C01827=1158.573,334.839,-76.760,-176.548,8.692,148.725
C01828=1158.569,335.087,-76.793,-176.546,8.695,148.726
C01829=1158.565,335.335,-76.827,-176.543,8.698,148.726
C01830=1158.562,335.582,-76.859,-176.540,8.702,148.726
C01831=1158.557,335.831,-76.892,-176.538,8.706,148.726
C01832=1158.553,336.078,-76.925,-176.536,8.709,148.726
C01833=1158.549,336.326,-76.958,-176.532,8.713,148.727
C01834=1158.545,336.574,-76.991,-176.530,8.716,148.727
C01835=1158.541,336.822,-77.024,-176.528,8.719,148.727
C01836=1158.537,337.069,-77.057,-176.525,8.723,148.727
C01837=1158.532,337.317,-77.091,-176.523,8.727,148.727
C01838=1158.529,337.565,-77.124,-176.520,8.730,148.728
C01839=1158.525,337.813,-77.157,-176.517,8.734,148.728
C01840=1158.521,338.061,-77.190,-176.515,8.737,148.728
C01841=1158.516,338.309,-77.224,-176.513,8.741,148.728
C01842=1158.512,338.556,-77.257,-176.510,8.745,148.728
C01843=1158.509,338.804,-77.291,-176.508,8.748,148.729
C01844=1158.504,339.051,-77.324,-176.505,8.751,148.729
C01845=1158.500,339.331,-77.361,-176.502,8.755,148.729
C01846=1158.495,339.612,-77.398,-176.500,8.759,148.729
C01847=1158.491,339.891,-77.436,-176.497,8.764,148.730
C01848=1158.486,340.171,-77.473,-176.494,8.768,148.730
C01849=1158.482,340.418,-77.508,-176.491,8.771,148.730
C01850=1158.478,340.666,-77.541,-176.489,8.775,148.730
C01851=1158.473,340.914,-77.574,-176.486,8.778,148.731
C01852=1158.469,341.162,-77.607,-176.484,8.782,148.731
C01853=1158.466,341.410,-77.641,-176.482,8.786,148.731
C01854=1158.462,341.657,-77.675,-176.479,8.789,148.731
C01855=1158.458,341.905,-77.708,-176.476,8.793,148.732
C01856=1158.454,342.153,-77.741,-176.474,8.797,148.732
C01857=1158.449,342.401,-77.775,-176.472,8.800,148.732
C01858=1158.445,342.648,-77.809,-176.469,8.804,148.732
C01859=1158.441,342.896,-77.842,-176.467,8.807,148.733
C01860=1158.437,343.144,-77.875,-176.464,8.811,148.733
C01861=1158.433,343.391,-77.909,-176.461,8.815,148.733
C01862=1158.429,343.639,-77.942,-176.459,8.818,148.733
C01863=1158.424,343.887,-77.976,-176.456,8.822,148.733
C01864=1158.421,344.135,-78.010,-176.454,8.825,148.734
C01865=1158.417,344.382,-78.044,-176.452,8.829,148.734
C01866=1158.413,344.629,-78.077,-176.449,8.833,148.734
C01867=1158.408,344.877,-78.111,-176.446,8.836,148.734
C01868=1158.405,345.124,-78.145,-176.444,8.841,148.735
C01869=1158.401,345.373,-78.179,-176.442,8.844,148.735
C01870=1158.397,345.621,-78.212,-176.439,8.847,148.735
C01871=1158.392,345.868,-78.246,-176.436,8.851,148.736
C01872=1158.388,346.116,-78.279,-176.434,8.854,148.736
C01873=1158.385,346.364,-78.314,-176.431,8.859,148.736
C01874=1158.381,346.611,-78.348,-176.429,8.862,148.736
C01875=1158.376,346.859,-78.381,-176.427,8.865,148.736
C01876=1158.372,347.106,-78.415,-176.424,8.869,148.737
C01877=1158.369,347.354,-78.449,-176.422,8.873,148.737
C01878=1158.364,347.602,-78.483,-176.419,8.877,148.737
C01879=1158.360,347.849,-78.516,-176.417,8.880,148.738
C01880=1158.357,348.097,-78.551,-176.414,8.884,148.738
C01881=1158.352,348.345,-78.585,-176.411,8.888,148.738
C01882=1158.348,348.592,-78.618,-176.409,8.891,148.738
C01883=1158.344,348.840,-78.652,-176.407,8.895,148.739
C01884=1158.340,349.088,-78.687,-176.404,8.899,148.739
C01885=1158.336,349.335,-78.720,-176.402,8.902,148.739
C01886=1158.332,349.583,-78.754,-176.399,8.906,148.739
C01887=1158.328,349.831,-78.789,-176.397,8.909,148.740
C01888=1158.324,350.078,-78.822,-176.394,8.913,148.740
C01889=1158.320,350.326,-78.856,-176.392,8.917,148.740
C01890=1158.316,350.574,-78.891,-176.389,8.921,148.740
C01891=1158.312,350.821,-78.925,-176.387,8.924,148.741
C01892=1158.308,351.068,-78.959,-176.385,8.928,148.741
C01893=1158.304,351.317,-78.993,-176.382,8.932,148.741
C01894=1158.300,351.564,-79.027,-176.380,8.935,148.742
C01895=1158.296,351.812,-79.062,-176.377,8.939,148.742
C01896=1158.292,352.059,-79.096,-176.375,8.943,148.742
C01897=1158.288,352.307,-79.130,-176.372,8.947,148.742
C01898=1158.284,352.554,-79.164,-176.369,8.950,148.743
C01899=1158.280,352.802,-79.199,-176.367,8.955,148.743
C01900=1158.276,353.050,-79.232,-176.365,8.958,148.743
C01901=1158.272,353.298,-79.267,-176.362,8.962,148.743
C01902=1158.268,353.545,-79.301,-176.359,8.965,148.744
C01903=1158.264,353.793,-79.335,-176.358,8.969,148.744
C01904=1158.260,354.040,-79.369,-176.355,8.973,148.744
C01905=1158.256,354.288,-79.404,-176.352,8.976,148.745
C01906=1158.252,354.535,-79.438,-176.350,8.980,148.745
C01907=1158.248,354.783,-79.473,-176.348,8.984,148.745
C01908=1158.244,355.031,-79.507,-176.345,8.988,148.746
C01909=1158.240,355.278,-79.541,-176.342,8.991,148.746
C01910=1158.236,355.526,-79.576,-176.340,8.995,148.746
C01911=1158.232,355.773,-79.610,-176.338,8.999,148.746
C01912=1158.228,356.021,-79.645,-176.335,9.003,148.747
C01913=1158.224,356.268,-79.680,-176.333,9.006,148.747
C01914=1158.221,356.516,-79.714,-176.330,9.011,148.747
C01915=1158.216,356.763,-79.749,-176.328,9.014,148.748
C01916=1158.212,357.011,-79.783,-176.325,9.018,148.748
C01917=1158.208,357.258,-79.817,-176.323,9.021,148.748
C01918=1158.204,357.507,-79.852,-176.320,9.026,148.749
C01919=1158.200,357.754,-79.887,-176.318,9.029,148.749
C01920=1158.197,358.001,-79.922,-176.315,9.033,148.749
C01921=1158.192,358.249,-79.956,-176.313,9.037,148.749
C01922=1158.188,358.497,-79.991,-176.310,9.041,148.750
C01923=1158.184,358.744,-80.025,-176.308,9.044,148.750
C01924=1158.181,358.991,-80.060,-176.305,9.049,148.750
C01925=1158.177,359.239,-80.095,-176.303,9.052,148.751
C01926=1158.172,359.487,-80.130,-176.300,9.056,148.751
C01927=1158.169,359.735,-80.164,-176.298,9.060,148.751
C01928=1158.165,359.982,-80.199,-176.295,9.064,148.752
C01929=1158.161,360.230,-80.234,-176.293,9.067,148.752
C01930=1158.156,360.477,-80.268,-176.291,9.071,148.752
C01931=1158.153,360.724,-80.303,-176.288,9.075,148.752
C01932=1158.149,360.972,-80.338,-176.285,9.079,148.753
C01933=1158.145,361.219,-80.373,-176.283,9.083,148.753
C01934=1158.141,361.467,-80.408,-176.281,9.086,148.753
C01935=1158.137,361.715,-80.443,-176.278,9.091,148.754
C01936=1158.133,361.962,-80.478,-176.276,9.094,148.754
C01937=1158.130,362.210,-80.512,-176.273,9.098,148.754
C01938=1158.125,362.457,-80.548,-176.271,9.103,148.755
C01939=1158.121,362.705,-80.582,-176.268,9.106,148.755
C01940=1158.117,362.952,-80.618,-176.266,9.110,148.756
C01941=1158.113,363.200,-80.652,-176.263,9.114,148.756
C01942=1158.109,363.447,-80.688,-176.261,9.118,148.756
C01943=1158.105,363.695,-80.722,-176.259,9.121,148.756
C01944=1158.102,363.942,-80.757,-176.256,9.125,148.757
C01945=1158.098,364.190,-80.792,-176.253,9.130,148.757
C01946=1158.094,364.437,-80.827,-176.251,9.133,148.757
C01947=1158.090,364.684,-80.863,-176.249,9.138,148.758
C01948=1158.086,364.933,-80.898,-176.246,9.141,148.758
C01949=1158.081,365.215,-80.938,-176.243,9.146,148.759
C01950=1158.077,365.498,-80.978,-176.241,9.150,148.759
C01951=1158.072,365.781,-81.019,-176.238,9.155,148.759
C01952=1158.068,366.063,-81.059,-176.235,9.159,148.760
C01953=1158.064,366.311,-81.094,-176.233,9.163,148.760
C01954=1158.060,366.558,-81.129,-176.231,9.167,148.761
C01955=1158.056,366.806,-81.164,-176.228,9.171,148.761
C01956=1158.053,367.053,-81.200,-176.226,9.175,148.761
C01957=1158.048,367.300,-81.235,-176.223,9.179,148.762
C01958=1158.044,367.548,-81.270,-176.221,9.183,148.762
C01959=1158.041,367.796,-81.305,-176.219,9.187,148.763
C01960=1158.037,368.043,-81.341,-176.216,9.191,148.763
C01961=1158.033,368.290,-81.376,-176.214,9.194,148.763
C01962=1158.029,368.537,-81.412,-176.212,9.199,148.764
C01963=1158.024,368.786,-81.447,-176.210,9.202,148.764
C01964=1158.021,369.033,-81.482,-176.208,9.207,148.765
C01965=1158.016,369.280,-81.518,-176.206,9.210,148.765
C01966=1158.013,369.528,-81.553,-176.203,9.215,148.765
C01967=1158.009,369.775,-81.589,-176.201,9.218,148.766
C01968=1158.005,370.023,-81.624,-176.198,9.223,148.766
C01969=1158.001,370.269,-81.660,-176.197,9.226,148.767
C01970=1157.998,370.517,-81.695,-176.194,9.231,148.767
C01971=1157.993,370.765,-81.731,-176.192,9.234,148.768
C01972=1157.989,371.013,-81.766,-176.190,9.238,148.768
C01973=1157.986,371.260,-81.802,-176.188,9.242,148.768
C01974=1157.981,371.507,-81.837,-176.186,9.246,148.769
C01975=1157.978,371.755,-81.872,-176.184,9.250,148.770
C01976=1157.974,372.002,-81.908,-176.182,9.254,148.770
C01977=1157.970,372.250,-81.944,-176.180,9.258,148.770
C01978=1157.966,372.497,-81.980,-176.178,9.262,148.771
C01979=1157.962,372.744,-82.016,-176.176,9.266,148.771
C01980=1157.958,372.991,-82.051,-176.174,9.270,148.772
C01981=1157.955,373.239,-82.087,-176.172,9.274,148.772
C01982=1157.950,373.486,-82.123,-176.171,9.278,148.773
C01983=1157.947,373.734,-82.158,-176.168,9.282,148.773
C01984=1157.943,373.981,-82.194,-176.166,9.286,148.774
C01985=1157.939,374.229,-82.229,-176.165,9.290,148.775
C01986=1157.935,374.477,-82.265,-176.163,9.293,148.775
C01987=1157.931,374.723,-82.301,-176.161,9.298,148.776
C01988=1157.927,374.970,-82.337,-176.159,9.302,148.776
C01989=1157.923,375.218,-82.373,-176.157,9.306,148.777
C01990=1157.919,375.466,-82.409,-176.156,9.309,148.777
C01991=1157.915,375.713,-82.444,-176.154,9.313,148.778
C01992=1157.911,375.960,-82.481,-176.152,9.318,148.778
C01993=1157.908,376.208,-82.517,-176.151,9.322,148.779
C01994=1157.904,376.455,-82.552,-176.149,9.325,148.779
C01995=1157.900,376.703,-82.588,-176.147,9.329,148.780
C01996=1157.896,376.949,-82.624,-176.146,9.333,148.781
C01997=1157.892,377.197,-82.660,-176.144,9.337,148.781
C01998=1157.888,377.445,-82.696,-176.143,9.341,148.782
C01999=1157.884,377.692,-82.731,-176.142,9.345,148.783
C02000=1157.881,377.939,-82.768,-176.140,9.349,148.783
C02001=1157.876,378.187,-82.804,-176.139,9.353,148.784
C02002=1157.873,378.434,-82.839,-176.137,9.356,148.784
C02003=1157.868,378.682,-82.876,-176.136,9.360,148.785
C02004=1157.865,378.929,-82.912,-176.134,9.364,148.786
C02005=1157.861,379.177,-82.947,-176.133,9.368,148.786
C02006=1157.857,379.424,-82.984,-176.132,9.372,148.787
C02007=1157.853,379.671,-83.020,-176.131,9.375,148.788
C02008=1157.849,379.919,-83.057,-176.129,9.379,148.788
C02009=1157.846,380.166,-83.092,-176.128,9.384,148.789
C02010=1157.841,380.413,-83.129,-176.127,9.387,148.790
C02011=1157.838,380.661,-83.165,-176.127,9.391,148.790
C02012=1157.833,380.909,-83.201,-176.125,9.395,148.791
C02013=1157.830,381.155,-83.237,-176.124,9.399,148.792
C02014=1157.826,381.403,-83.272,-176.123,9.402,148.793
C02015=1157.822,381.650,-83.309,-176.122,9.406,148.793
C02016=1157.819,381.898,-83.345,-176.121,9.409,148.794
C02017=1157.815,382.145,-83.382,-176.120,9.413,148.795
C02018=1157.811,382.392,-83.417,-176.120,9.417,148.795
C02019=1157.807,382.639,-83.454,-176.118,9.421,148.796
C02020=1157.803,382.887,-83.490,-176.118,9.424,148.797
C02021=1157.799,383.134,-83.527,-176.117,9.428,148.798
C02022=1157.795,383.382,-83.562,-176.116,9.432,148.798
C02023=1157.791,383.629,-83.599,-176.116,9.435,148.799
C02024=1157.788,383.876,-83.635,-176.115,9.439,148.800
C02025=1157.784,384.124,-83.671,-176.115,9.442,148.801
C02026=1157.779,384.371,-83.708,-176.114,9.446,148.801
C02027=1157.776,384.618,-83.744,-176.114,9.449,148.802
C02028=1157.772,384.865,-83.781,-176.113,9.453,148.803
C02029=1157.768,385.113,-83.816,-176.113,9.456,148.804
C02030=1157.764,385.360,-83.853,-176.112,9.460,148.805
C02031=1157.761,385.607,-83.889,-176.112,9.463,148.805
C02032=1157.756,385.855,-83.925,-176.111,9.466,148.806
C02033=1157.753,386.102,-83.962,-176.111,9.469,148.807
C02034=1157.749,386.349,-83.999,-176.111,9.473,148.808
C02035=1157.744,386.597,-84.035,-176.111,9.476,148.809
C02036=1157.741,386.844,-84.071,-176.110,9.479,148.809
C02037=1157.737,387.091,-84.108,-176.111,9.482,148.810
C02038=1157.733,387.338,-84.143,-176.111,9.486,148.811
C02039=1157.729,387.585,-84.180,-176.111,9.488,148.812
C02040=1157.726,387.832,-84.216,-176.111,9.492,148.813
C02041=1157.721,388.080,-84.253,-176.111,9.495,148.813
C02042=1157.717,388.327,-84.289,-176.111,9.498,148.814
C02043=1157.714,388.574,-84.326,-176.111,9.501,148.815
C02044=1157.709,388.822,-84.362,-176.110,9.504,148.816
C02045=1157.707,389.070,-84.399,-176.111,9.507,148.817
C02046=1157.703,389.317,-84.435,-176.111,9.510,148.817
C02047=1157.698,389.565,-84.472,-176.111,9.513,148.818
C02048=1157.695,389.811,-84.508,-176.112,9.516,148.819
C02049=1157.691,390.059,-84.545,-176.112,9.519,148.820
C02050=1157.687,390.306,-84.582,-176.112,9.522,148.821
C02051=1157.683,390.553,-84.617,-176.112,9.524,148.822
C02052=1157.679,390.801,-84.654,-176.113,9.527,148.823
C02053=1157.675,391.086,-84.696,-176.113,9.531,148.823
C02054=1157.671,391.372,-84.738,-176.114,9.534,148.824
C02055=1157.666,391.659,-84.780,-176.114,9.537,148.825
C02056=1157.662,391.944,-84.822,-176.114,9.541,148.826
C02057=1157.658,392.191,-84.859,-176.115,9.543,148.827
C02058=1157.653,392.439,-84.895,-176.116,9.545,148.828
C02059=1157.650,392.686,-84.932,-176.116,9.548,148.829
C02060=1157.646,392.933,-84.969,-176.116,9.551,148.830
C02061=1157.642,393.181,-85.006,-176.117,9.553,148.830
C02062=1157.638,393.428,-85.041,-176.117,9.556,148.831
C02063=1157.634,393.675,-85.078,-176.118,9.558,148.832
C02064=1157.630,393.922,-85.115,-176.119,9.561,148.833
C02065=1157.627,394.169,-85.151,-176.119,9.564,148.834
C02066=1157.623,394.417,-85.188,-176.119,9.566,148.835
C02067=1157.618,394.664,-85.224,-176.121,9.568,148.835
C02068=1157.615,394.911,-85.261,-176.121,9.571,148.836
C02069=1157.611,395.158,-85.297,-176.122,9.573,148.837
C02070=1157.608,395.406,-85.335,-176.122,9.576,148.838
C02071=1157.604,395.653,-85.371,-176.122,9.579,148.839
C02072=1157.600,395.901,-85.407,-176.124,9.581,148.839
C02073=1157.596,396.148,-85.444,-176.124,9.583,148.840
C02074=1157.592,396.395,-85.480,-176.125,9.585,148.841
C02075=1157.588,396.642,-85.517,-176.125,9.588,148.842
C02076=1157.584,396.889,-85.554,-176.126,9.590,148.843
C02077=1157.580,397.137,-85.589,-176.127,9.592,148.843
C02078=1157.576,397.384,-85.626,-176.127,9.594,148.844
C02079=1157.572,397.631,-85.663,-176.128,9.597,148.845
C02080=1157.570,397.879,-85.700,-176.129,9.599,148.846
C02081=1157.565,398.126,-85.737,-176.130,9.601,148.846
C02082=1157.561,398.374,-85.773,-176.131,9.603,148.847
C02083=1157.558,398.621,-85.809,-176.131,9.606,148.848
C02084=1157.554,398.868,-85.846,-176.132,9.608,148.849
C02085=1157.549,399.115,-85.883,-176.133,9.610,148.849
C02086=1157.546,399.362,-85.919,-176.133,9.612,148.850
C02087=1157.542,399.609,-85.956,-176.134,9.614,148.851
C02088=1157.538,399.857,-85.992,-176.135,9.616,148.852
C02089=1157.534,400.104,-86.029,-176.136,9.618,148.853
C02090=1157.531,400.352,-86.066,-176.136,9.621,148.853
C02091=1157.527,400.599,-86.102,-176.137,9.623,148.854
C02092=1157.523,400.846,-86.139,-176.138,9.625,148.855
C02093=1157.519,401.093,-86.176,-176.139,9.626,148.856
C02094=1157.515,401.341,-86.212,-176.140,9.628,148.856
C02095=1157.511,401.588,-86.249,-176.140,9.631,148.857
C02096=1157.507,401.835,-86.285,-176.141,9.633,148.858
C02097=1157.503,402.082,-86.322,-176.142,9.635,148.859
C02098=1157.499,402.329,-86.359,-176.143,9.637,148.859
C02099=1157.496,402.577,-86.396,-176.144,9.639,148.860
C02100=1157.492,402.825,-86.431,-176.144,9.640,148.861
C02101=1157.488,403.072,-86.468,-176.145,9.643,148.861
C02102=1157.484,403.319,-86.505,-176.146,9.645,148.862
C02103=1157.480,403.566,-86.541,-176.146,9.647,148.863
C02104=1157.476,403.813,-86.578,-176.147,9.649,148.864
C02105=1157.472,404.060,-86.615,-176.148,9.650,148.864
C02106=1157.468,404.308,-86.652,-176.149,9.652,148.865
C02107=1157.465,404.556,-86.688,-176.150,9.654,148.866
C02108=1157.461,404.803,-86.725,-176.150,9.656,148.866
C02109=1157.457,405.050,-86.761,-176.151,9.658,148.867
C02110=1157.454,405.297,-86.798,-176.152,9.660,148.868
C02111=1157.449,405.544,-86.835,-176.152,9.662,148.869
C02112=1157.445,405.791,-86.871,-176.153,9.664,148.869
C02113=1157.442,406.038,-86.908,-176.154,9.666,148.870
C02114=1157.438,406.286,-86.944,-176.155,9.668,148.871
C02115=1157.434,406.534,-86.981,-176.155,9.670,148.871
C02116=1157.430,406.781,-87.018,-176.156,9.671,148.872
C02117=1157.427,407.028,-87.054,-176.157,9.673,148.873
C02118=1157.423,407.275,-87.091,-176.157,9.675,148.873
C02119=1157.419,407.522,-87.128,-176.158,9.677,148.874
C02120=1157.415,407.769,-87.164,-176.159,9.678,148.875
C02121=1157.411,408.017,-87.200,-176.160,9.680,148.875
C02122=1157.407,408.264,-87.237,-176.161,9.682,148.876
C02123=1157.403,408.512,-87.274,-176.161,9.684,148.877
C02124=1157.400,408.759,-87.311,-176.162,9.686,148.877
C02125=1157.396,409.006,-87.348,-176.162,9.688,148.878
C02126=1157.392,409.253,-87.384,-176.163,9.690,148.879
C02127=1157.388,409.500,-87.421,-176.164,9.692,148.879
C02128=1157.384,409.748,-87.458,-176.164,9.693,148.880
C02129=1157.380,409.995,-87.494,-176.165,9.695,148.881
C02130=1157.376,410.243,-87.531,-176.166,9.697,148.881
C02131=1157.373,410.490,-87.567,-176.166,9.699,148.882
C02132=1157.369,410.737,-87.604,-176.167,9.700,148.883
C02133=1157.365,410.985,-87.641,-176.168,9.702,148.883
C02134=1157.361,411.232,-87.678,-176.168,9.704,148.884
C02135=1157.357,411.479,-87.714,-176.169,9.706,148.884
C02136=1157.353,411.726,-87.751,-176.170,9.707,148.885
C02137=1157.349,411.973,-87.788,-176.170,9.709,148.886
C02138=1157.345,412.221,-87.824,-176.170,9.711,148.886
C02139=1157.342,412.468,-87.860,-176.171,9.713,148.887
C02140=1157.338,412.716,-87.897,-176.172,9.715,148.888
C02141=1157.334,412.963,-87.934,-176.172,9.717,148.888
C02142=1157.330,413.210,-87.970,-176.173,9.718,148.889
C02143=1157.326,413.457,-88.007,-176.174,9.720,148.889
C02144=1157.322,413.704,-88.044,-176.174,9.722,148.890
C02145=1157.318,413.951,-88.081,-176.175,9.724,148.891
C02146=1157.315,414.198,-88.117,-176.175,9.725,148.891
C02147=1157.311,414.446,-88.155,-176.175,9.728,148.892
C02148=1157.307,414.694,-88.191,-176.176,9.729,148.893
C02149=1157.303,414.941,-88.228,-176.177,9.731,148.893
C02150=1157.299,415.188,-88.264,-176.177,9.733,148.894
C02151=1157.297,415.435,-88.301,-176.178,9.734,148.894
C02152=1157.296,415.683,-88.338,-176.178,9.736,148.895
C02153=1157.294,416.068,-88.394,-176.179,9.739,148.896
C02154=1157.295,416.454,-88.451,-176.179,9.742,148.897
C02155=1157.298,416.840,-88.507,-176.181,9.744,148.898
C02156=1157.303,417.224,-88.562,-176.181,9.747,148.898
C02157=1156.882,417.227,-88.610,-176.184,9.758,148.902
C02158=1156.878,416.838,-88.553,-176.183,9.756,148.901
C02159=1156.875,416.450,-88.497,-176.183,9.753,148.900
C02160=1156.873,416.060,-88.440,-176.182,9.750,148.900
C02161=1156.875,415.671,-88.382,-176.181,9.747,148.898
C02162=1156.877,415.424,-88.346,-176.181,9.745,148.898
C02163=1156.879,415.177,-88.310,-176.180,9.744,148.897
C02164=1156.882,414.929,-88.273,-176.179,9.742,148.897
C02165=1156.886,414.681,-88.236,-176.179,9.740,148.896
C02166=1156.890,414.435,-88.200,-176.178,9.738,148.895
C02167=1156.894,414.187,-88.163,-176.178,9.737,148.895
C02168=1156.898,413.940,-88.126,-176.178,9.734,148.894
C02169=1156.902,413.693,-88.089,-176.177,9.733,148.894
C02170=1156.905,413.445,-88.053,-176.176,9.731,148.893
C02171=1156.909,413.198,-88.016,-176.176,9.729,148.892
C02172=1156.913,412.951,-87.979,-176.175,9.727,148.892
C02173=1156.917,412.704,-87.942,-176.174,9.726,148.891
C02174=1156.920,412.457,-87.906,-176.174,9.724,148.890
C02175=1156.925,412.209,-87.870,-176.173,9.722,148.890
C02176=1156.929,411.962,-87.833,-176.173,9.721,148.889
C02177=1156.933,411.715,-87.796,-176.172,9.719,148.889
C02178=1156.936,411.467,-87.759,-176.172,9.716,148.888
C02179=1156.940,411.220,-87.723,-176.171,9.715,148.887
C02180=1156.944,410.973,-87.686,-176.170,9.713,148.887
C02181=1156.948,410.726,-87.649,-176.170,9.711,148.886
C02182=1156.951,410.479,-87.613,-176.169,9.709,148.885
C02183=1156.956,410.232,-87.576,-176.168,9.708,148.885
C02184=1156.960,409.984,-87.539,-176.168,9.706,148.884
C02185=1156.963,409.736,-87.503,-176.167,9.704,148.883
C02186=1156.967,409.489,-87.466,-176.166,9.702,148.883
C02187=1156.971,409.242,-87.429,-176.166,9.701,148.882
C02188=1156.975,408.995,-87.392,-176.165,9.699,148.882
C02189=1156.978,408.748,-87.356,-176.164,9.697,148.881
C02190=1156.982,408.500,-87.319,-176.164,9.695,148.880
C02191=1156.986,408.253,-87.282,-176.162,9.693,148.879
C02192=1156.991,408.006,-87.246,-176.162,9.692,148.879
C02193=1156.993,407.759,-87.209,-176.161,9.690,148.878
C02194=1156.998,407.511,-87.173,-176.161,9.687,148.877
C02195=1157.002,407.264,-87.136,-176.160,9.685,148.877
C02196=1157.005,407.017,-87.100,-176.160,9.684,148.876
C02197=1157.009,406.769,-87.063,-176.159,9.682,148.876
C02198=1157.013,406.522,-87.026,-176.158,9.680,148.875
C02199=1157.017,406.275,-86.989,-176.157,9.678,148.874
C02200=1157.021,406.028,-86.953,-176.156,9.676,148.873
C02201=1157.024,405.780,-86.916,-176.156,9.675,148.873
C02202=1157.029,405.532,-86.879,-176.155,9.673,148.872
C02203=1157.032,405.286,-86.843,-176.154,9.671,148.871
C02204=1157.036,405.038,-86.806,-176.153,9.669,148.871
C02205=1157.040,404.791,-86.769,-176.152,9.667,148.870
C02206=1157.044,404.544,-86.733,-176.152,9.666,148.869
C02207=1157.048,404.297,-86.696,-176.151,9.664,148.868
C02208=1157.052,404.050,-86.659,-176.151,9.661,148.868
C02209=1157.055,403.802,-86.622,-176.150,9.659,148.867
C02210=1157.059,403.555,-86.587,-176.149,9.657,148.866
C02211=1157.063,403.307,-86.550,-176.148,9.655,148.866
C02212=1157.067,403.060,-86.513,-176.147,9.654,148.865
C02213=1157.071,402.813,-86.476,-176.146,9.652,148.864
C02214=1157.075,402.566,-86.440,-176.145,9.650,148.863
C02215=1157.079,402.319,-86.403,-176.145,9.648,148.863
C02216=1157.083,402.072,-86.366,-176.144,9.646,148.862
C02217=1157.086,401.824,-86.330,-176.144,9.643,148.861
C02218=1157.090,401.576,-86.293,-176.142,9.641,148.860
C02219=1157.094,401.329,-86.257,-176.142,9.640,148.860
C02220=1157.098,401.082,-86.220,-176.141,9.638,148.859
C02221=1157.102,400.835,-86.183,-176.140,9.636,148.858
C02222=1157.106,400.588,-86.147,-176.139,9.633,148.857
C02223=1157.110,400.341,-86.110,-176.139,9.631,148.857
C02224=1157.113,400.093,-86.074,-176.138,9.629,148.856
C02225=1157.117,399.845,-86.037,-176.137,9.627,148.855
C02226=1157.121,399.598,-86.000,-176.136,9.625,148.854
C02227=1157.125,399.351,-85.963,-176.136,9.623,148.854
C02228=1157.128,399.104,-85.927,-176.135,9.621,148.853
C02229=1157.132,398.857,-85.890,-176.134,9.619,148.852
C02230=1157.137,398.609,-85.854,-176.133,9.616,148.851
C02231=1157.140,398.362,-85.818,-176.133,9.614,148.851
C02232=1157.144,398.115,-85.781,-176.131,9.612,148.850
C02233=1157.148,397.868,-85.744,-176.131,9.610,148.849
C02234=1157.151,397.620,-85.707,-176.130,9.608,148.848
C02235=1157.155,397.373,-85.670,-176.129,9.606,148.847
C02236=1157.160,397.125,-85.634,-176.129,9.603,148.847
C02237=1157.163,396.878,-85.598,-176.128,9.601,148.846
C02238=1157.167,396.631,-85.561,-176.127,9.598,148.845
C02239=1157.171,396.384,-85.524,-176.127,9.596,148.844
C02240=1157.175,396.137,-85.487,-176.126,9.594,148.843
C02241=1157.179,395.889,-85.452,-176.125,9.592,148.843
C02242=1157.183,395.642,-85.415,-176.125,9.589,148.842
C02243=1157.187,395.395,-85.378,-176.124,9.587,148.841
C02244=1157.190,395.147,-85.342,-176.124,9.584,148.840
C02245=1157.194,394.900,-85.305,-176.122,9.582,148.840
C02246=1157.198,394.653,-85.268,-176.122,9.579,148.839
C02247=1157.202,394.405,-85.232,-176.121,9.578,148.838
C02248=1157.206,394.158,-85.195,-176.121,9.575,148.837
C02249=1157.210,393.911,-85.159,-176.120,9.572,148.836
C02250=1157.213,393.664,-85.122,-176.120,9.569,148.835
C02251=1157.217,393.417,-85.085,-176.119,9.567,148.835
C02252=1157.222,393.169,-85.049,-176.118,9.564,148.834
C02253=1157.225,392.922,-85.013,-176.118,9.562,148.833
C02254=1157.229,392.674,-84.976,-176.118,9.559,148.832
C02255=1157.233,392.427,-84.939,-176.116,9.557,148.831
C02256=1157.236,392.180,-84.903,-176.116,9.554,148.831
C02257=1157.241,391.933,-84.867,-176.116,9.551,148.830
C02258=1157.245,391.647,-84.824,-176.115,9.549,148.829
C02259=1157.249,391.361,-84.783,-176.115,9.545,148.828
C02260=1157.254,391.075,-84.740,-176.115,9.542,148.827
C02261=1157.259,390.789,-84.697,-176.114,9.539,148.826
C02262=1157.262,390.542,-84.661,-176.114,9.536,148.825
C02263=1157.266,390.294,-84.625,-176.114,9.533,148.824
C02264=1157.270,390.048,-84.589,-176.114,9.530,148.823
C02265=1157.274,389.800,-84.552,-176.113,9.527,148.823
C02266=1157.277,389.552,-84.515,-176.112,9.524,148.822
C02267=1157.281,389.305,-84.479,-176.112,9.522,148.821
C02268=1157.285,389.058,-84.442,-176.112,9.518,148.820
C02269=1157.289,388.811,-84.405,-176.112,9.515,148.819
C02270=1157.293,388.564,-84.369,-176.112,9.512,148.818
C02271=1157.297,388.316,-84.333,-176.112,9.509,148.818
C02272=1157.300,388.069,-84.297,-176.112,9.506,148.817
C02273=1157.304,387.822,-84.260,-176.112,9.503,148.816
C02274=1157.309,387.574,-84.224,-176.112,9.500,148.815
C02275=1157.312,387.327,-84.187,-176.112,9.497,148.814
C02276=1157.316,387.080,-84.151,-176.112,9.494,148.814
C02277=1157.320,386.832,-84.115,-176.112,9.490,148.813
C02278=1157.324,386.585,-84.078,-176.112,9.487,148.812
C02279=1157.328,386.338,-84.041,-176.112,9.484,148.811
C02280=1157.332,386.091,-84.006,-176.113,9.481,148.810
C02281=1157.335,385.843,-83.969,-176.113,9.477,148.809
C02282=1157.339,385.596,-83.932,-176.113,9.474,148.809
C02283=1157.343,385.348,-83.896,-176.114,9.471,148.808
C02284=1157.346,385.101,-83.860,-176.114,9.467,148.807
C02285=1157.350,384.854,-83.823,-176.114,9.464,148.806
C02286=1157.355,384.606,-83.787,-176.115,9.460,148.806
C02287=1157.358,384.359,-83.751,-176.115,9.457,148.805
C02288=1157.363,384.111,-83.715,-176.116,9.454,148.804
C02289=1157.366,383.865,-83.678,-176.116,9.450,148.803
C02290=1157.370,383.617,-83.641,-176.117,9.446,148.802
C02291=1157.374,383.370,-83.606,-176.118,9.443,148.802
C02292=1157.378,383.123,-83.569,-176.118,9.439,148.801
C02293=1157.381,382.875,-83.533,-176.119,9.435,148.800
C02294=1157.386,382.628,-83.497,-176.120,9.432,148.800
C02295=1157.389,382.380,-83.461,-176.121,9.429,148.799
C02296=1157.393,382.133,-83.424,-176.122,9.424,148.798
C02297=1157.397,381.886,-83.389,-176.122,9.421,148.797
C02298=1157.401,381.639,-83.352,-176.124,9.417,148.797
C02299=1157.405,381.391,-83.316,-176.125,9.413,148.796
C02300=1157.409,381.144,-83.279,-176.125,9.410,148.795
C02301=1157.412,380.896,-83.244,-176.126,9.406,148.794
C02302=1157.417,380.649,-83.207,-176.127,9.403,148.794
C02303=1157.420,380.402,-83.171,-176.128,9.398,148.793
C02304=1157.424,380.155,-83.135,-176.130,9.394,148.792
C02305=1157.428,379.907,-83.099,-176.131,9.391,148.792
C02306=1157.432,379.660,-83.062,-176.132,9.387,148.791
C02307=1157.436,379.412,-83.027,-176.133,9.383,148.790
C02308=1157.439,379.165,-82.991,-176.135,9.379,148.790
C02309=1157.444,378.918,-82.954,-176.136,9.375,148.789
C02310=1157.447,378.670,-82.919,-176.137,9.371,148.788
C02311=1157.452,378.422,-82.883,-176.139,9.367,148.788
C02312=1157.456,378.176,-82.847,-176.140,9.363,148.787
C02313=1157.459,377.929,-82.811,-176.141,9.360,148.786
C02314=1157.464,377.681,-82.775,-176.143,9.356,148.786
C02315=1157.467,377.434,-82.739,-176.144,9.352,148.785
C02316=1157.471,377.186,-82.703,-176.146,9.348,148.785
C02317=1157.475,376.939,-82.667,-176.148,9.344,148.784
C02318=1157.478,376.692,-82.631,-176.149,9.340,148.783
C02319=1157.483,376.444,-82.595,-176.151,9.336,148.783
C02320=1157.486,376.196,-82.559,-176.152,9.333,148.782
C02321=1157.490,375.949,-82.523,-176.154,9.329,148.782
C02322=1157.494,375.702,-82.487,-176.156,9.324,148.781
C02323=1157.498,375.454,-82.451,-176.157,9.320,148.781
C02324=1157.502,375.207,-82.416,-176.159,9.316,148.780
C02325=1157.507,374.960,-82.380,-176.161,9.313,148.779
C02326=1157.510,374.713,-82.343,-176.163,9.308,148.779
C02327=1157.514,374.465,-82.308,-176.165,9.305,148.778
C02328=1157.518,374.217,-82.272,-176.166,9.301,148.778
C02329=1157.522,373.970,-82.236,-176.168,9.297,148.777
C02330=1157.525,373.722,-82.201,-176.170,9.292,148.777
C02331=1157.529,373.475,-82.165,-176.172,9.289,148.776
C02332=1157.534,373.228,-82.129,-176.174,9.285,148.776
C02333=1157.537,372.981,-82.093,-176.176,9.280,148.775
C02334=1157.541,372.733,-82.058,-176.178,9.277,148.775
C02335=1157.545,372.486,-82.022,-176.180,9.273,148.774
C02336=1157.548,372.238,-81.986,-176.182,9.269,148.774
C02337=1157.553,371.991,-81.950,-176.184,9.265,148.773
C02338=1157.557,371.744,-81.915,-176.186,9.261,148.773
C02339=1157.561,371.496,-81.880,-176.188,9.257,148.772
C02340=1157.564,371.249,-81.844,-176.190,9.253,148.772
C02341=1157.568,371.001,-81.808,-176.192,9.249,148.771
C02342=1157.572,370.754,-81.772,-176.194,9.245,148.771
C02343=1157.577,370.507,-81.737,-176.197,9.241,148.771
C02344=1157.580,370.259,-81.702,-176.198,9.237,148.770
C02345=1157.584,370.012,-81.666,-176.201,9.233,148.770
C02346=1157.588,369.764,-81.631,-176.203,9.229,148.769
C02347=1157.592,369.516,-81.596,-176.205,9.225,148.769
C02348=1157.596,369.269,-81.561,-176.207,9.221,148.768
C02349=1157.599,369.022,-81.525,-176.210,9.217,148.768
C02350=1157.604,368.774,-81.489,-176.212,9.214,148.768
C02351=1157.608,368.527,-81.453,-176.214,9.209,148.767
C02352=1157.612,368.280,-81.418,-176.216,9.206,148.767
C02353=1157.615,368.032,-81.383,-176.219,9.201,148.766
C02354=1157.619,367.784,-81.348,-176.222,9.197,148.766
C02355=1157.623,367.537,-81.312,-176.223,9.194,148.766
C02356=1157.627,367.290,-81.277,-176.226,9.189,148.765
C02357=1157.631,367.042,-81.241,-176.228,9.186,148.765
C02358=1157.635,366.794,-81.207,-176.231,9.182,148.764
C02359=1157.639,366.547,-81.171,-176.233,9.178,148.764
C02360=1157.643,366.300,-81.136,-176.235,9.174,148.764
C02361=1157.647,366.052,-81.100,-176.237,9.170,148.763
C02362=1157.652,365.770,-81.060,-176.240,9.165,148.763
C02363=1157.656,365.486,-81.020,-176.243,9.161,148.762
C02364=1157.661,365.203,-80.980,-176.246,9.156,148.762
C02365=1157.665,364.921,-80.940,-176.248,9.152,148.762
C02366=1157.669,364.674,-80.905,-176.251,9.148,148.761
C02367=1157.672,364.426,-80.869,-176.254,9.144,148.761
C02368=1157.677,364.179,-80.835,-176.256,9.140,148.761
C02369=1157.680,363.931,-80.799,-176.258,9.136,148.760
C02370=1157.684,363.683,-80.764,-176.261,9.133,148.760
C02371=1157.689,363.436,-80.729,-176.263,9.128,148.759
C02372=1157.693,363.188,-80.694,-176.266,9.124,148.759
C02373=1157.696,362.941,-80.659,-176.268,9.121,148.759
C02374=1157.700,362.693,-80.625,-176.271,9.116,148.758
C02375=1157.704,362.446,-80.589,-176.273,9.113,148.758
C02376=1157.708,362.199,-80.555,-176.276,9.109,148.758
C02377=1157.712,361.951,-80.519,-176.278,9.105,148.758
C02378=1157.716,361.703,-80.484,-176.281,9.101,148.757
C02379=1157.720,361.456,-80.449,-176.283,9.097,148.757
C02380=1157.723,361.208,-80.415,-176.285,9.094,148.757
C02381=1157.728,360.961,-80.380,-176.288,9.089,148.756
C02382=1157.732,360.713,-80.345,-176.290,9.086,148.756
C02383=1157.736,360.465,-80.310,-176.293,9.082,148.756
C02384=1157.740,360.218,-80.275,-176.295,9.078,148.755
C02385=1157.743,359.971,-80.241,-176.298,9.074,148.755
C02386=1157.748,359.723,-80.206,-176.301,9.070,148.755
C02387=1157.751,359.476,-80.171,-176.303,9.066,148.754
C02388=1157.756,359.228,-80.136,-176.306,9.062,148.754
C02389=1157.759,358.980,-80.102,-176.308,9.059,148.754
C02390=1157.763,358.733,-80.066,-176.310,9.055,148.753
C02391=1157.767,358.486,-80.032,-176.313,9.051,148.753
C02392=1157.771,358.238,-79.998,-176.316,9.047,148.753
C02393=1157.775,357.990,-79.963,-176.317,9.044,148.752
C02394=1157.779,357.742,-79.928,-176.320,9.040,148.752
C02395=1157.783,357.495,-79.893,-176.323,9.036,148.752
C02396=1157.787,357.248,-79.859,-176.325,9.032,148.752
C02397=1157.791,357.000,-79.825,-176.327,9.029,148.751
C02398=1157.795,356.752,-79.790,-176.330,9.024,148.751
C02399=1157.799,356.505,-79.756,-176.333,9.021,148.751
C02400=1157.803,356.257,-79.721,-176.335,9.017,148.750
C02401=1157.807,356.010,-79.686,-176.337,9.013,148.750
C02402=1157.811,355.762,-79.652,-176.340,9.009,148.750
C02403=1157.815,355.515,-79.617,-176.342,9.006,148.749
C02404=1157.818,355.267,-79.583,-176.345,9.002,148.749
C02405=1157.823,355.020,-79.548,-176.347,8.998,148.749
C02406=1157.827,354.771,-79.514,-176.350,8.994,148.749
C02407=1157.831,354.524,-79.480,-176.352,8.991,148.748
C02408=1157.835,354.277,-79.445,-176.355,8.987,148.748
C02409=1157.839,354.029,-79.411,-176.357,8.983,148.748
C02410=1157.843,353.782,-79.377,-176.360,8.979,148.747
C02411=1157.846,353.534,-79.342,-176.362,8.976,148.747
C02412=1157.851,353.286,-79.308,-176.365,8.972,148.747
C02413=1157.854,353.039,-79.274,-176.367,8.968,148.747
C02414=1157.859,352.791,-79.239,-176.370,8.965,148.746
C02415=1157.863,352.544,-79.205,-176.372,8.961,148.746
C02416=1157.867,352.295,-79.171,-176.374,8.957,148.746
C02417=1157.871,352.048,-79.137,-176.377,8.953,148.745
C02418=1157.875,351.800,-79.102,-176.379,8.950,148.745
C02419=1157.879,351.553,-79.068,-176.382,8.946,148.745
C02420=1157.883,351.306,-79.034,-176.384,8.942,148.745
C02421=1157.886,351.058,-79.000,-176.387,8.938,148.744
C02422=1157.891,350.810,-78.966,-176.389,8.935,148.744
C02423=1157.895,350.563,-78.932,-176.392,8.931,148.744
C02424=1157.899,350.315,-78.897,-176.395,8.927,148.744
C02425=1157.903,350.067,-78.864,-176.397,8.924,148.743
C02426=1157.907,349.820,-78.829,-176.399,8.920,148.743
C02427=1157.911,349.572,-78.796,-176.402,8.916,148.743
C02428=1157.915,349.324,-78.762,-176.405,8.912,148.742
C02429=1157.919,349.077,-78.727,-176.407,8.909,148.742
C02430=1157.923,348.829,-78.694,-176.409,8.905,148.742
C02431=1157.927,348.581,-78.659,-176.412,8.901,148.742
C02432=1157.931,348.334,-78.625,-176.414,8.898,148.741
C02433=1157.935,348.086,-78.592,-176.417,8.894,148.741
C02434=1157.939,347.838,-78.557,-176.419,8.891,148.741
C02435=1157.943,347.591,-78.524,-176.422,8.887,148.741
C02436=1157.947,347.343,-78.490,-176.424,8.883,148.740
C02437=1157.951,347.095,-78.456,-176.427,8.879,148.740
C02438=1157.955,346.848,-78.422,-176.429,8.876,148.740
C02439=1157.959,346.600,-78.389,-176.431,8.872,148.740
C02440=1157.963,346.352,-78.354,-176.434,8.868,148.739
C02441=1157.967,346.105,-78.321,-176.437,8.865,148.739
C02442=1157.971,345.857,-78.287,-176.440,8.861,148.739
C02443=1157.976,345.609,-78.253,-176.442,8.858,148.739
C02444=1157.980,345.361,-78.219,-176.444,8.854,148.738
C02445=1157.983,345.114,-78.186,-176.447,8.850,148.738
C02446=1157.988,344.866,-78.152,-176.449,8.847,148.738
C02447=1157.992,344.619,-78.118,-176.452,8.842,148.738
C02448=1157.996,344.370,-78.084,-176.454,8.839,148.737
C02449=1157.999,344.123,-78.051,-176.456,8.836,148.737
C02450=1158.004,343.875,-78.017,-176.459,8.832,148.737
C02451=1158.008,343.628,-77.984,-176.462,8.829,148.737
C02452=1158.012,343.380,-77.950,-176.464,8.824,148.736
C02453=1158.016,343.132,-77.916,-176.467,8.821,148.736
C02454=1158.020,342.885,-77.882,-176.469,8.818,148.736
C02455=1158.024,342.637,-77.849,-176.472,8.814,148.736
C02456=1158.028,342.389,-77.816,-176.474,8.810,148.735
C02457=1158.033,342.141,-77.782,-176.476,8.807,148.735
C02458=1158.037,341.894,-77.748,-176.479,8.803,148.735
C02459=1158.040,341.646,-77.715,-176.481,8.799,148.735
C02460=1158.044,341.398,-77.682,-176.484,8.795,148.734
C02461=1158.048,341.151,-77.648,-176.487,8.792,148.734
C02462=1158.052,340.903,-77.615,-176.489,8.789,148.734
C02463=1158.056,340.655,-77.582,-176.492,8.785,148.734
C02464=1158.061,340.408,-77.548,-176.494,8.781,148.734
C02465=1158.065,340.160,-77.515,-176.496,8.778,148.733
C02466=1158.069,339.879,-77.477,-176.499,8.774,148.733
C02467=1158.074,339.600,-77.439,-176.502,8.770,148.733
C02468=1158.079,339.320,-77.402,-176.505,8.766,148.733
C02469=1158.083,339.041,-77.364,-176.508,8.762,148.732
C02470=1158.087,338.793,-77.331,-176.510,8.758,148.732
C02471=1158.091,338.544,-77.297,-176.513,8.754,148.732
C02472=1158.095,338.297,-77.264,-176.515,8.751,148.732
C02473=1158.099,338.049,-77.231,-176.518,8.747,148.731
C02474=1158.103,337.801,-77.198,-176.521,8.744,148.731
C02475=1158.107,337.554,-77.165,-176.523,8.740,148.731
C02476=1158.111,337.306,-77.131,-176.526,8.736,148.731
C02477=1158.115,337.059,-77.098,-176.528,8.733,148.731
C02478=1158.120,336.811,-77.065,-176.530,8.730,148.730
C02479=1158.124,336.563,-77.032,-176.533,8.726,148.730
C02480=1158.128,336.315,-76.999,-176.536,8.722,148.730
C02481=1158.132,336.067,-76.966,-176.538,8.719,148.730
C02482=1158.136,335.819,-76.933,-176.541,8.715,148.729
C02483=1158.141,335.572,-76.900,-176.543,8.712,148.729
C02484=1158.145,335.324,-76.866,-176.545,8.708,148.729
C02485=1158.148,335.077,-76.834,-176.548,8.704,148.729
C02486=1158.152,334.829,-76.801,-176.551,8.701,148.729
C02487=1158.156,334.580,-76.767,-176.553,8.698,148.728
C02488=1158.160,334.333,-76.734,-176.556,8.694,148.728
C02489=1158.164,334.085,-76.701,-176.559,8.691,148.728
C02490=1158.169,333.837,-76.668,-176.561,8.687,148.728
C02491=1158.173,333.589,-76.635,-176.564,8.683,148.728
C02492=1158.176,333.341,-76.603,-176.566,8.680,148.727
C02493=1158.181,333.094,-76.570,-176.568,8.677,148.727
C02494=1158.185,332.847,-76.537,-176.571,8.673,148.727
C02495=1158.189,332.598,-76.504,-176.574,8.669,148.727
C02496=1158.194,332.351,-76.471,-176.576,8.666,148.727
C02497=1158.197,332.103,-76.439,-176.578,8.663,148.726
C02498=1158.201,331.856,-76.405,-176.581,8.659,148.726
C02499=1158.206,331.607,-76.373,-176.583,8.655,148.726
C02500=1158.210,331.359,-76.340,-176.586,8.652,148.726
C02501=1158.213,331.112,-76.307,-176.589,8.648,148.726
C02502=1158.217,330.864,-76.275,-176.591,8.645,148.726
C02503=1158.222,330.616,-76.242,-176.594,8.642,148.725
C02504=1158.226,330.368,-76.209,-176.596,8.638,148.725
C02505=1158.229,330.120,-76.177,-176.599,8.634,148.725
C02506=1158.234,329.872,-76.144,-176.601,8.631,148.725
C02507=1158.238,329.624,-76.111,-176.603,8.628,148.725
C02508=1158.242,329.376,-76.078,-176.606,8.624,148.724
C02509=1158.246,329.129,-76.046,-176.609,8.621,148.724
C02510=1158.251,328.881,-76.013,-176.611,8.617,148.724
C02511=1158.255,328.634,-75.980,-176.614,8.613,148.724
C02512=1158.258,328.386,-75.948,-176.617,8.610,148.724
C02513=1158.263,328.138,-75.915,-176.619,8.607,148.723
C02514=1158.267,327.889,-75.883,-176.621,8.603,148.723
C02515=1158.271,327.641,-75.851,-176.624,8.599,148.723
C02516=1158.275,327.394,-75.818,-176.627,8.596,148.723
C02517=1158.279,327.146,-75.786,-176.629,8.593,148.723
C02518=1158.283,326.899,-75.753,-176.631,8.590,148.723
C02519=1158.288,326.650,-75.721,-176.634,8.586,148.722
C02520=1158.291,326.403,-75.688,-176.637,8.582,148.722
C02521=1158.296,326.154,-75.656,-176.639,8.579,148.722
C02522=1158.299,325.906,-75.624,-176.642,8.575,148.722
C02523=1158.304,325.659,-75.591,-176.645,8.572,148.722
C02524=1158.308,325.411,-75.559,-176.647,8.569,148.722
C02525=1158.312,325.163,-75.527,-176.649,8.566,148.721
C02526=1158.316,324.916,-75.494,-176.652,8.561,148.721
C02527=1158.320,324.667,-75.462,-176.655,8.558,148.721
C02528=1158.324,324.419,-75.430,-176.657,8.555,148.721
C02529=1158.329,324.172,-75.397,-176.659,8.552,148.721
C02530=1158.332,323.924,-75.365,-176.662,8.548,148.721
C02531=1158.337,323.676,-75.333,-176.665,8.545,148.720
C02532=1158.340,323.428,-75.301,-176.667,8.542,148.720
C02533=1158.345,323.181,-75.268,-176.670,8.538,148.720
C02534=1158.349,322.933,-75.236,-176.673,8.534,148.720
C02535=1158.353,322.684,-75.204,-176.675,8.531,148.720
C02536=1158.357,322.436,-75.172,-176.678,8.528,148.720
C02537=1158.361,322.188,-75.140,-176.680,8.525,148.720
C02538=1158.365,321.941,-75.107,-176.683,8.521,148.719
C02539=1158.369,321.693,-75.076,-176.685,8.517,148.719
C02540=1158.374,321.445,-75.043,-176.687,8.514,148.719
C02541=1158.377,321.197,-75.011,-176.690,8.511,148.719
C02542=1158.382,320.949,-74.979,-176.693,8.507,148.719
C02543=1158.386,320.701,-74.947,-176.695,8.504,148.718
C02544=1158.390,320.453,-74.916,-176.698,8.500,148.718
C02545=1158.395,320.205,-74.883,-176.700,8.497,148.718
C02546=1158.398,319.957,-74.852,-176.703,8.493,148.718
C02547=1158.402,319.709,-74.820,-176.706,8.490,148.718
C02548=1158.407,319.461,-74.787,-176.708,8.487,148.718
C02549=1158.411,319.214,-74.756,-176.711,8.484,148.718
C02550=1158.415,318.966,-74.724,-176.713,8.480,148.718
C02551=1158.419,318.717,-74.692,-176.716,8.476,148.717
C02552=1158.423,318.470,-74.660,-176.719,8.473,148.717
C02553=1158.427,318.222,-74.628,-176.721,8.470,148.717
C02554=1158.431,317.974,-74.596,-176.723,8.467,148.717
C02555=1158.436,317.726,-74.564,-176.726,8.463,148.717
C02556=1158.440,317.478,-74.532,-176.729,8.460,148.717
C02557=1158.443,317.230,-74.501,-176.731,8.457,148.716
C02558=1158.448,316.983,-74.469,-176.733,8.453,148.716
C02559=1158.452,316.734,-74.437,-176.736,8.450,148.716
C02560=1158.457,316.486,-74.406,-176.739,8.446,148.716
C02561=1158.460,316.238,-74.374,-176.741,8.443,148.716
C02562=1158.464,315.990,-74.342,-176.744,8.440,148.716
C02563=1158.469,315.743,-74.310,-176.746,8.437,148.716
C02564=1158.473,315.495,-74.278,-176.749,8.433,148.716
C02565=1158.477,315.246,-74.247,-176.752,8.430,148.716
C02566=1158.481,314.999,-74.216,-176.754,8.426,148.715
C02567=1158.485,314.751,-74.184,-176.757,8.423,148.715
C02568=1158.489,314.503,-74.152,-176.759,8.420,148.715
C02569=1158.494,314.254,-74.121,-176.762,8.417,148.715
C02570=1158.499,313.978,-74.085,-176.765,8.413,148.715
C02571=1158.503,313.700,-74.050,-176.768,8.409,148.715
C02572=1158.508,313.423,-74.015,-176.771,8.405,148.714
C02573=1158.512,313.146,-73.979,-176.773,8.401,148.714
C02574=1158.517,312.898,-73.948,-176.776,8.399,148.714
C02575=1158.521,312.650,-73.916,-176.779,8.394,148.714
C02576=1158.524,312.402,-73.885,-176.782,8.391,148.714
C02577=1158.529,312.154,-73.854,-176.784,8.388,148.714
C02578=1158.533,311.906,-73.822,-176.786,8.385,148.714
C02579=1158.537,311.658,-73.791,-176.789,8.382,148.714
C02580=1158.541,311.410,-73.759,-176.792,8.378,148.714
C02581=1158.546,311.162,-73.729,-176.794,8.375,148.713
C02582=1158.549,310.914,-73.697,-176.797,8.372,148.713
C02583=1158.554,310.666,-73.666,-176.799,8.368,148.713
C02584=1158.558,310.418,-73.634,-176.802,8.365,148.713
C02585=1158.562,310.170,-73.603,-176.804,8.362,148.713
C02586=1158.566,309.922,-73.571,-176.807,8.358,148.713
C02587=1158.571,309.674,-73.541,-176.810,8.355,148.713
C02588=1158.574,309.426,-73.509,-176.812,8.352,148.713
C02589=1158.579,309.178,-73.478,-176.815,8.349,148.713
C02590=1158.583,308.930,-73.447,-176.817,8.345,148.712
C02591=1158.587,308.682,-73.415,-176.819,8.342,148.712
C02592=1158.592,308.434,-73.384,-176.823,8.338,148.712
C02593=1158.596,308.186,-73.353,-176.825,8.335,148.712
C02594=1158.600,307.938,-73.322,-176.828,8.332,148.712
C02595=1158.604,307.690,-73.290,-176.830,8.329,148.712
C02596=1158.608,307.442,-73.260,-176.832,8.326,148.712
C02597=1158.612,307.193,-73.228,-176.835,8.323,148.712
C02598=1158.617,306.946,-73.197,-176.838,8.319,148.711
C02599=1158.621,306.698,-73.166,-176.841,8.316,148.712
C02600=1158.625,306.449,-73.136,-176.843,8.312,148.711
C02601=1158.629,306.202,-73.105,-176.846,8.309,148.711
C02602=1158.633,305.953,-73.073,-176.848,8.306,148.711
C02603=1158.638,305.706,-73.042,-176.851,8.303,148.711
C02604=1158.642,305.458,-73.011,-176.853,8.300,148.711
C02605=1158.646,305.209,-72.980,-176.856,8.296,148.711
C02606=1158.651,304.962,-72.949,-176.859,8.293,148.711
C02607=1158.654,304.714,-72.919,-176.861,8.289,148.711
C02608=1158.658,304.465,-72.888,-176.864,8.286,148.711
C02609=1158.663,304.217,-72.857,-176.866,8.283,148.710
C02610=1158.667,303.969,-72.826,-176.869,8.280,148.711
C02611=1158.672,303.721,-72.795,-176.871,8.277,148.710
C02612=1158.676,303.473,-72.765,-176.875,8.273,148.710
C02613=1158.679,303.225,-72.733,-176.877,8.270,148.710
C02614=1158.684,302.977,-72.702,-176.880,8.267,148.710
C02615=1158.688,302.729,-72.671,-176.882,8.264,148.710
C02616=1158.692,302.481,-72.641,-176.885,8.261,148.710
C02617=1158.696,302.233,-72.610,-176.887,8.257,148.710
C02618=1158.701,301.985,-72.579,-176.890,8.254,148.710
C02619=1158.706,301.737,-72.549,-176.892,8.251,148.710
C02620=1158.709,301.489,-72.518,-176.896,8.247,148.710
C02621=1158.713,301.241,-72.487,-176.898,8.244,148.709
C02622=1158.718,300.993,-72.456,-176.901,8.241,148.710
C02623=1158.721,300.744,-72.426,-176.903,8.238,148.709
C02624=1158.726,300.496,-72.395,-176.906,8.235,148.709
C02625=1158.731,300.248,-72.364,-176.908,8.232,148.709
C02626=1158.734,300.001,-72.334,-176.911,8.229,148.709
C02627=1158.738,299.752,-72.303,-176.913,8.225,148.709
C02628=1158.743,299.503,-72.273,-176.916,8.222,148.709
C02629=1158.747,299.256,-72.243,-176.919,8.218,148.709
C02630=1158.752,299.008,-72.212,-176.921,8.215,148.709
C02631=1158.756,298.759,-72.181,-176.924,8.212,148.709
C02632=1158.760,298.512,-72.151,-176.926,8.209,148.709
C02633=1158.764,298.264,-72.120,-176.929,8.206,148.709
C02634=1158.768,298.016,-72.090,-176.932,8.203,148.709
C02635=1158.773,297.767,-72.059,-176.934,8.200,148.708
C02636=1158.776,297.519,-72.029,-176.937,8.197,148.708
C02637=1158.781,297.271,-71.999,-176.939,8.193,148.708
C02638=1158.786,297.023,-71.968,-176.942,8.190,148.708
C02639=1158.790,296.775,-71.938,-176.945,8.187,148.708
C02640=1158.794,296.526,-71.907,-176.947,8.183,148.708
C02641=1158.798,296.279,-71.877,-176.950,8.180,148.708
C02642=1158.802,296.031,-71.846,-176.952,8.177,148.708
C02643=1158.807,295.782,-71.817,-176.955,8.174,148.708
C02644=1158.811,295.534,-71.786,-176.957,8.171,148.708
C02645=1158.814,295.286,-71.756,-176.960,8.168,148.708
C02646=1158.819,295.037,-71.725,-176.963,8.165,148.708
C02647=1158.823,294.790,-71.695,-176.965,8.162,148.708
C02648=1158.827,294.542,-71.665,-176.968,8.159,148.708
C02649=1158.832,294.294,-71.635,-176.970,8.155,148.708
C02650=1158.836,294.046,-71.605,-176.974,8.152,148.708
C02651=1158.840,293.797,-71.574,-176.976,8.149,148.708
C02652=1158.844,293.549,-71.544,-176.979,8.145,148.707
C02653=1158.849,293.301,-71.514,-176.981,8.142,148.707
C02654=1158.853,293.053,-71.484,-176.984,8.139,148.707
C02655=1158.857,292.805,-71.454,-176.987,8.136,148.707
C02656=1158.862,292.557,-71.424,-176.989,8.133,148.707
C02657=1158.866,292.309,-71.394,-176.992,8.130,148.707
C02658=1158.870,292.061,-71.364,-176.994,8.127,148.707
C02659=1158.874,291.812,-71.333,-176.997,8.124,148.707
C02660=1158.878,291.564,-71.304,-176.999,8.121,148.707
C02661=1158.883,291.316,-71.273,-177.002,8.118,148.707
C02662=1158.887,291.067,-71.243,-177.004,8.115,148.707
C02663=1158.891,290.819,-71.214,-177.007,8.112,148.707
C02664=1158.896,290.571,-71.183,-177.011,8.108,148.707
C02665=1158.900,290.323,-71.154,-177.013,8.105,148.707
C02666=1158.904,290.075,-71.124,-177.016,8.102,148.707
C02667=1158.908,289.827,-71.094,-177.018,8.098,148.707
C02668=1158.913,289.578,-71.064,-177.021,8.095,148.707
C02669=1158.917,289.331,-71.034,-177.023,8.092,148.707
C02670=1158.921,289.083,-71.004,-177.026,8.089,148.707
C02671=1158.925,288.834,-70.975,-177.029,8.086,148.707
C02672=1158.930,288.586,-70.944,-177.031,8.083,148.707
C02673=1158.934,288.338,-70.915,-177.034,8.080,148.706
C02674=1158.939,288.063,-70.882,-177.037,8.076,148.706
C02675=1158.943,287.787,-70.849,-177.040,8.073,148.706
C02676=1158.948,287.512,-70.816,-177.042,8.070,148.707
C02677=1158.952,287.237,-70.783,-177.045,8.066,148.706
C02678=1158.956,286.989,-70.753,-177.048,8.063,148.706
C02679=1158.961,286.741,-70.724,-177.051,8.060,148.706
C02680=1158.965,286.493,-70.694,-177.053,8.057,148.706
C02681=1158.969,286.244,-70.663,-177.056,8.054,148.706
C02682=1158.974,285.996,-70.634,-177.059,8.051,148.706
C02683=1158.978,285.748,-70.605,-177.061,8.048,148.706
C02684=1158.983,285.500,-70.576,-177.064,8.045,148.706
C02685=1158.987,285.252,-70.546,-177.066,8.042,148.706
C02686=1158.991,285.004,-70.517,-177.069,8.039,148.706
C02687=1158.995,284.755,-70.487,-177.072,8.036,148.706
C02688=1159.000,284.507,-70.456,-177.074,8.033,148.706
C02689=1159.004,284.259,-70.427,-177.077,8.030,148.706
C02690=1159.008,284.011,-70.397,-177.079,8.026,148.706
C02691=1159.012,283.763,-70.368,-177.082,8.023,148.706
C02692=1159.016,283.514,-70.339,-177.085,8.020,148.706
C02693=1159.021,283.266,-70.309,-177.087,8.017,148.706
C02694=1159.025,283.018,-70.280,-177.090,8.014,148.706
C02695=1159.029,282.770,-70.250,-177.093,8.011,148.706
C02696=1159.033,282.521,-70.221,-177.095,8.008,148.706
C02697=1159.038,282.274,-70.192,-177.098,8.005,148.706
C02698=1159.042,282.025,-70.162,-177.101,8.001,148.706
C02699=1159.047,281.777,-70.133,-177.104,7.998,148.706
C02700=1159.051,281.528,-70.104,-177.107,7.995,148.706
C02701=1159.055,281.280,-70.075,-177.109,7.992,148.706
C02702=1159.059,281.032,-70.045,-177.112,7.989,148.706
C02703=1159.063,280.783,-70.016,-177.114,7.986,148.706
C02704=1159.068,280.535,-69.986,-177.117,7.983,148.706
C02705=1159.072,280.288,-69.957,-177.120,7.980,148.706
C02706=1159.077,280.039,-69.928,-177.122,7.977,148.706
C02707=1159.081,279.791,-69.899,-177.125,7.974,148.706
C02708=1159.085,279.542,-69.869,-177.128,7.971,148.706
C02709=1159.089,279.294,-69.840,-177.130,7.968,148.706
C02710=1159.094,279.046,-69.811,-177.133,7.965,148.706
C02711=1159.098,278.798,-69.781,-177.136,7.962,148.706
C02712=1159.103,278.549,-69.753,-177.138,7.959,148.706
C02713=1159.106,278.301,-69.724,-177.141,7.956,148.706
C02714=1159.110,278.053,-69.694,-177.143,7.954,148.706
C02715=1159.115,277.804,-69.666,-177.146,7.951,148.706
C02716=1159.120,277.557,-69.637,-177.148,7.948,148.706
C02717=1159.124,277.308,-69.607,-177.151,7.945,148.706
C02718=1159.128,277.060,-69.578,-177.153,7.941,148.706
C02719=1159.133,276.811,-69.549,-177.156,7.938,148.706
C02720=1159.136,276.563,-69.520,-177.159,7.935,148.706
C02721=1159.141,276.315,-69.492,-177.162,7.932,148.706
C02722=1159.145,276.067,-69.462,-177.165,7.930,148.706
C02723=1159.149,275.818,-69.433,-177.167,7.926,148.706
C02724=1159.154,275.570,-69.404,-177.170,7.923,148.706
C02725=1159.158,275.322,-69.376,-177.172,7.920,148.706
C02726=1159.162,275.073,-69.347,-177.175,7.917,148.706
C02727=1159.167,274.825,-69.317,-177.178,7.914,148.706
C02728=1159.171,274.577,-69.288,-177.181,7.912,148.706
C02729=1159.175,274.329,-69.260,-177.183,7.908,148.706
C02730=1159.179,274.081,-69.231,-177.186,7.905,148.706
C02731=1159.184,273.832,-69.202,-177.188,7.902,148.706
C02732=1159.188,273.584,-69.173,-177.191,7.899,148.706
C02733=1159.192,273.336,-69.145,-177.194,7.896,148.706
C02734=1159.197,273.087,-69.116,-177.197,7.893,148.706
C02735=1159.201,272.839,-69.087,-177.199,7.890,148.706
C02736=1159.205,272.591,-69.059,-177.202,7.887,148.706
C02737=1159.210,272.342,-69.029,-177.205,7.884,148.706
C02738=1159.214,272.094,-69.001,-177.207,7.881,148.706
C02739=1159.218,271.846,-68.972,-177.210,7.878,148.706
C02740=1159.223,271.597,-68.943,-177.213,7.875,148.706
C02741=1159.227,271.349,-68.915,-177.215,7.872,148.706
C02742=1159.231,271.101,-68.886,-177.218,7.869,148.706
C02743=1159.236,270.852,-68.857,-177.221,7.866,148.706
C02744=1159.240,270.603,-68.829,-177.223,7.864,148.706
C02745=1159.244,270.356,-68.800,-177.226,7.861,148.706
C02746=1159.249,270.107,-68.771,-177.228,7.858,148.706
C02747=1159.252,269.859,-68.743,-177.231,7.855,148.706
C02748=1159.258,269.611,-68.715,-177.234,7.852,148.706
C02749=1159.262,269.362,-68.685,-177.236,7.849,148.706
C02750=1159.266,269.114,-68.658,-177.239,7.846,148.706
C02751=1159.271,268.866,-68.629,-177.242,7.843,148.706
C02752=1159.274,268.617,-68.601,-177.245,7.840,148.706
C02753=1159.279,268.369,-68.572,-177.247,7.837,148.706
C02754=1159.283,268.121,-68.544,-177.250,7.834,148.706
C02755=1159.288,267.873,-68.515,-177.253,7.831,148.707
C02756=1159.292,267.624,-68.487,-177.256,7.828,148.707
C02757=1159.297,267.376,-68.459,-177.258,7.825,148.707
C02758=1159.300,267.127,-68.431,-177.261,7.822,148.707
C02759=1159.305,266.879,-68.401,-177.263,7.820,148.707
C02760=1159.309,266.631,-68.373,-177.266,7.817,148.707
C02761=1159.314,266.382,-68.345,-177.268,7.814,148.707
C02762=1159.318,266.134,-68.317,-177.271,7.811,148.707
C02763=1159.322,265.886,-68.288,-177.274,7.808,148.707
C02764=1159.327,265.638,-68.260,-177.277,7.805,148.707
C02765=1159.331,265.389,-68.232,-177.279,7.802,148.707
C02766=1159.336,265.141,-68.204,-177.282,7.799,148.707
C02767=1159.340,264.892,-68.175,-177.285,7.796,148.707
C02768=1159.344,264.644,-68.147,-177.288,7.793,148.707
C02769=1159.348,264.396,-68.119,-177.290,7.790,148.707
C02770=1159.353,264.147,-68.091,-177.293,7.788,148.707
C02771=1159.357,263.899,-68.063,-177.295,7.785,148.707
C02772=1159.362,263.651,-68.034,-177.298,7.782,148.707
C02773=1159.366,263.402,-68.006,-177.301,7.779,148.707
C02774=1159.370,263.154,-67.978,-177.303,7.776,148.707
C02775=1159.375,262.905,-67.950,-177.306,7.773,148.707
C02776=1159.379,262.657,-67.922,-177.309,7.770,148.707
C02777=1159.383,262.408,-67.894,-177.312,7.767,148.707
C02778=1159.388,262.135,-67.862,-177.314,7.764,148.707
C02779=1159.393,261.862,-67.832,-177.317,7.761,148.708
C02780=1159.397,261.588,-67.801,-177.321,7.758,148.708
C02781=1159.403,261.316,-67.771,-177.324,7.755,148.708
C02782=1159.406,261.067,-67.743,-177.326,7.752,148.708
C02783=1159.412,260.819,-67.714,-177.329,7.749,148.708
C02784=1159.416,260.570,-67.687,-177.332,7.746,148.708
C02785=1159.420,260.322,-67.659,-177.334,7.744,148.708
C02786=1159.424,260.073,-67.631,-177.336,7.741,148.708
C02787=1159.429,259.825,-67.602,-177.339,7.738,148.708
C02788=1159.433,259.577,-67.575,-177.342,7.735,148.708
C02789=1159.437,259.328,-67.547,-177.345,7.732,148.708
C02790=1159.442,259.080,-67.519,-177.348,7.729,148.708
C02791=1159.446,258.831,-67.491,-177.350,7.726,148.708
C02792=1159.451,258.583,-67.464,-177.353,7.723,148.708
C02793=1159.455,258.335,-67.436,-177.355,7.721,148.708
C02794=1159.459,258.086,-67.408,-177.358,7.718,148.708
C02795=1159.463,257.838,-67.381,-177.361,7.715,148.709
C02796=1159.467,257.589,-67.353,-177.364,7.713,148.709
C02797=1159.473,257.341,-67.325,-177.367,7.710,148.709
C02798=1159.477,257.093,-67.297,-177.370,7.707,148.709
C02799=1159.481,256.844,-67.270,-177.372,7.704,148.709
C02800=1159.485,256.596,-67.242,-177.374,7.702,148.709
C02801=1159.490,256.348,-67.214,-177.377,7.699,148.709
C02802=1159.494,256.099,-67.187,-177.380,7.696,148.709
C02803=1159.498,255.851,-67.159,-177.383,7.693,148.709
C02804=1159.504,255.602,-67.131,-177.386,7.690,148.709
C02805=1159.507,255.353,-67.103,-177.388,7.687,148.709
C02806=1159.512,255.105,-67.076,-177.391,7.684,148.709
C02807=1159.516,254.857,-67.048,-177.393,7.682,148.710
C02808=1159.520,254.608,-67.021,-177.396,7.679,148.710
C02809=1159.525,254.360,-66.993,-177.399,7.676,148.710
C02810=1159.529,254.111,-66.966,-177.402,7.673,148.710
C02811=1159.534,253.863,-66.939,-177.404,7.670,148.710
C02812=1159.538,253.614,-66.911,-177.407,7.667,148.710
C02813=1159.542,253.366,-66.884,-177.409,7.665,148.710
C02814=1159.547,253.118,-66.856,-177.412,7.662,148.710
C02815=1159.551,252.869,-66.829,-177.415,7.659,148.710
C02816=1159.555,252.620,-66.802,-177.418,7.656,148.710
C02817=1159.560,252.372,-66.774,-177.420,7.653,148.710
C02818=1159.564,252.124,-66.747,-177.424,7.650,148.710
C02819=1159.569,251.875,-66.719,-177.426,7.648,148.711
C02820=1159.573,251.627,-66.691,-177.429,7.645,148.711
C02821=1159.578,251.378,-66.664,-177.431,7.642,148.711
C02822=1159.582,251.130,-66.637,-177.434,7.640,148.711
C02823=1159.586,250.881,-66.609,-177.437,7.637,148.711
C02824=1159.591,250.633,-66.582,-177.440,7.634,148.711
C02825=1159.595,250.384,-66.555,-177.442,7.632,148.711
C02826=1159.600,250.136,-66.528,-177.445,7.629,148.711
C02827=1159.604,249.888,-66.501,-177.447,7.626,148.711
C02828=1159.608,249.639,-66.473,-177.450,7.623,148.711
C02829=1159.612,249.390,-66.446,-177.453,7.620,148.712
C02830=1159.617,249.142,-66.419,-177.456,7.618,148.712
C02831=1159.622,248.893,-66.392,-177.458,7.615,148.712
C02832=1159.626,248.645,-66.365,-177.461,7.612,148.712
C02833=1159.631,248.397,-66.337,-177.464,7.609,148.712
C02834=1159.635,248.148,-66.310,-177.467,7.606,148.712
C02835=1159.639,247.900,-66.283,-177.469,7.604,148.712
C02836=1159.643,247.651,-66.256,-177.472,7.601,148.712
C02837=1159.648,247.403,-66.229,-177.475,7.598,148.712
C02838=1159.653,247.154,-66.202,-177.478,7.596,148.712
C02839=1159.657,246.906,-66.175,-177.480,7.593,148.712
C02840=1159.660,246.657,-66.148,-177.483,7.590,148.713
C02841=1159.665,246.408,-66.121,-177.485,7.588,148.713
C02842=1159.670,246.160,-66.094,-177.488,7.585,148.713
C02843=1159.674,245.911,-66.067,-177.491,7.582,148.713
C02844=1159.679,245.663,-66.040,-177.494,7.579,148.713
C02845=1159.683,245.415,-66.014,-177.496,7.577,148.713
C02846=1159.688,245.166,-65.987,-177.499,7.574,148.713
C02847=1159.692,244.918,-65.960,-177.502,7.571,148.713
C02848=1159.697,244.669,-65.933,-177.505,7.568,148.713
C02849=1159.700,244.420,-65.906,-177.507,7.565,148.713
C02850=1159.705,244.172,-65.879,-177.510,7.563,148.714
C02851=1159.710,243.923,-65.852,-177.513,7.560,148.714
C02852=1159.714,243.675,-65.825,-177.516,7.557,148.714
C02853=1159.718,243.427,-65.798,-177.518,7.554,148.714
C02854=1159.723,243.178,-65.771,-177.521,7.552,148.714
C02855=1159.727,242.929,-65.745,-177.523,7.549,148.714
C02856=1159.732,242.681,-65.718,-177.526,7.546,148.714
C02857=1159.736,242.432,-65.691,-177.529,7.544,148.715
C02858=1159.740,242.184,-65.665,-177.532,7.542,148.715
C02859=1159.745,241.936,-65.638,-177.534,7.539,148.715
C02860=1159.750,241.687,-65.611,-177.537,7.536,148.715
C02861=1159.754,241.438,-65.585,-177.540,7.533,148.715
C02862=1159.759,241.190,-65.558,-177.542,7.531,148.715
C02863=1159.762,240.942,-65.531,-177.545,7.528,148.715
C02864=1159.767,240.693,-65.505,-177.548,7.525,148.715
C02865=1159.772,240.444,-65.478,-177.551,7.522,148.715
C02866=1159.776,240.196,-65.451,-177.553,7.520,148.715
C02867=1159.781,239.947,-65.424,-177.556,7.518,148.716
C02868=1159.785,239.699,-65.399,-177.559,7.515,148.716
C02869=1159.790,239.450,-65.371,-177.562,7.512,148.716
C02870=1159.793,239.202,-65.345,-177.564,7.510,148.716
C02871=1159.798,238.953,-65.319,-177.567,7.507,148.716
C02872=1159.802,238.705,-65.292,-177.570,7.504,148.716
C02873=1159.807,238.456,-65.266,-177.573,7.501,148.716
C02874=1159.811,238.207,-65.239,-177.575,7.499,148.717
C02875=1159.816,237.959,-65.212,-177.578,7.496,148.717
C02876=1159.820,237.710,-65.187,-177.581,7.493,148.717
C02877=1159.825,237.462,-65.160,-177.584,7.490,148.717
C02878=1159.829,237.213,-65.134,-177.586,7.488,148.717
C02879=1159.834,236.964,-65.107,-177.589,7.485,148.717
C02880=1159.838,236.715,-65.081,-177.591,7.482,148.717
C02881=1159.843,236.467,-65.054,-177.594,7.481,148.718
C02882=1159.847,236.196,-65.025,-177.597,7.477,148.718
C02883=1159.852,235.923,-64.997,-177.600,7.474,148.718
C02884=1159.857,235.652,-64.968,-177.603,7.471,148.718
C02885=1159.862,235.380,-64.939,-177.606,7.468,148.718
C02886=1159.866,235.132,-64.913,-177.608,7.466,148.718
C02887=1159.870,234.883,-64.887,-177.612,7.464,148.719
C02888=1159.876,234.635,-64.860,-177.614,7.461,148.719
C02889=1159.880,234.386,-64.834,-177.617,7.458,148.719
C02890=1159.885,234.137,-64.808,-177.619,7.456,148.719
C02891=1159.889,233.889,-64.782,-177.623,7.453,148.719
C02892=1159.893,233.640,-64.756,-177.625,7.450,148.719
C02893=1159.898,233.392,-64.729,-177.628,7.448,148.719
C02894=1159.902,233.143,-64.703,-177.631,7.445,148.720
C02895=1159.907,232.895,-64.678,-177.634,7.443,148.720
C02896=1159.911,232.646,-64.651,-177.636,7.440,148.720
C02897=1159.915,232.398,-64.625,-177.639,7.437,148.720
C02898=1159.920,232.149,-64.599,-177.642,7.435,148.720
C02899=1159.925,231.900,-64.573,-177.644,7.433,148.720
C02900=1159.929,231.651,-64.546,-177.647,7.430,148.720
C02901=1159.933,231.403,-64.521,-177.650,7.427,148.721
C02902=1159.938,231.155,-64.495,-177.653,7.424,148.721
C02903=1159.943,230.905,-64.469,-177.655,7.422,148.721
C02904=1159.946,230.657,-64.442,-177.658,7.419,148.721
C02905=1159.951,230.408,-64.417,-177.661,7.417,148.721
C02906=1159.956,230.160,-64.391,-177.663,7.414,148.721
C02907=1159.961,229.911,-64.365,-177.666,7.412,148.721
C02908=1159.965,229.662,-64.339,-177.669,7.409,148.722
C02909=1159.969,229.414,-64.313,-177.671,7.407,148.722
C02910=1159.973,229.165,-64.287,-177.674,7.404,148.722
C02911=1159.978,228.917,-64.262,-177.677,7.401,148.722
C02912=1159.983,228.668,-64.235,-177.680,7.399,148.722
C02913=1159.987,228.419,-64.209,-177.682,7.396,148.722
C02914=1159.991,228.171,-64.184,-177.686,7.394,148.723
C02915=1159.996,227.922,-64.158,-177.688,7.391,148.723
C02916=1160.000,227.674,-64.133,-177.691,7.389,148.723
C02917=1160.004,227.425,-64.107,-177.694,7.386,148.723
C02918=1160.009,227.176,-64.081,-177.696,7.384,148.723
C02919=1160.014,226.928,-64.055,-177.699,7.381,148.723
C02920=1160.018,226.679,-64.029,-177.702,7.379,148.724
C02921=1160.023,226.430,-64.004,-177.704,7.376,148.724
C02922=1160.027,226.182,-63.978,-177.707,7.373,148.724
C02923=1160.032,225.933,-63.952,-177.710,7.371,148.724
C02924=1160.036,225.684,-63.927,-177.713,7.369,148.724
C02925=1160.041,225.436,-63.901,-177.715,7.366,148.724
C02926=1160.045,225.187,-63.876,-177.718,7.364,148.725
C02927=1160.049,224.939,-63.850,-177.721,7.361,148.725
C02928=1160.053,224.690,-63.824,-177.724,7.358,148.725
C02929=1160.058,224.442,-63.799,-177.726,7.356,148.725
C02930=1160.062,224.193,-63.773,-177.729,7.353,148.725
C02931=1160.067,223.944,-63.747,-177.731,7.351,148.725
C02932=1160.072,223.696,-63.722,-177.734,7.349,148.726
C02933=1160.076,223.447,-63.697,-177.737,7.346,148.726
C02934=1160.081,223.198,-63.671,-177.740,7.344,148.726
C02935=1160.085,222.950,-63.646,-177.743,7.341,148.726
C02936=1160.089,222.701,-63.620,-177.745,7.338,148.726
C02937=1160.094,222.453,-63.594,-177.748,7.336,148.727
C02938=1160.099,222.203,-63.569,-177.751,7.333,148.727
C02939=1160.103,221.955,-63.544,-177.753,7.331,148.727
C02940=1160.108,221.706,-63.518,-177.756,7.328,148.727
C02941=1160.112,221.458,-63.493,-177.759,7.326,148.727
C02942=1160.117,221.209,-63.468,-177.762,7.324,148.728
C02943=1160.121,220.960,-63.442,-177.765,7.321,148.728
C02944=1160.126,220.711,-63.416,-177.767,7.319,148.728
C02945=1160.130,220.463,-63.391,-177.770,7.316,148.728
C02946=1160.135,220.214,-63.366,-177.773,7.313,148.728
C02947=1160.140,219.966,-63.341,-177.775,7.311,148.729
C02948=1160.144,219.717,-63.315,-177.778,7.308,148.729
C02949=1160.148,219.468,-63.290,-177.780,7.306,148.729
C02950=1160.153,219.220,-63.265,-177.784,7.304,148.729
C02951=1160.157,218.971,-63.239,-177.786,7.301,148.729
C02952=1160.162,218.722,-63.215,-177.789,7.299,148.729
C02953=1160.166,218.473,-63.189,-177.792,7.296,148.730
C02954=1160.171,218.225,-63.164,-177.794,7.294,148.730
C02955=1160.175,217.976,-63.139,-177.797,7.291,148.730
C02956=1160.180,217.727,-63.114,-177.800,7.289,148.730
C02957=1160.184,217.479,-63.089,-177.803,7.287,148.730
C02958=1160.189,217.230,-63.063,-177.806,7.284,148.730
C02959=1160.193,216.981,-63.038,-177.808,7.282,148.731
C02960=1160.198,216.733,-63.013,-177.811,7.279,148.731
C02961=1160.202,216.484,-62.988,-177.813,7.277,148.731
C02962=1160.207,216.236,-62.963,-177.816,7.274,148.731
C02963=1160.211,215.986,-62.938,-177.819,7.272,148.731
C02964=1160.216,215.738,-62.914,-177.822,7.270,148.732
C02965=1160.220,215.489,-62.888,-177.825,7.267,148.732
C02966=1160.225,215.240,-62.863,-177.827,7.265,148.732
C02967=1160.229,214.992,-62.838,-177.830,7.262,148.732
C02968=1160.234,214.743,-62.814,-177.833,7.260,148.733
C02969=1160.238,214.494,-62.788,-177.836,7.257,148.733
C02970=1160.243,214.246,-62.763,-177.838,7.255,148.733
C02971=1160.247,213.996,-62.739,-177.841,7.253,148.733
C02972=1160.252,213.748,-62.713,-177.843,7.250,148.733
C02973=1160.256,213.499,-62.688,-177.846,7.248,148.734
C02974=1160.261,213.251,-62.664,-177.849,7.246,148.734
C02975=1160.265,213.002,-62.638,-177.852,7.243,148.734
C02976=1160.270,212.753,-62.614,-177.854,7.241,148.734
C02977=1160.274,212.505,-62.590,-177.857,7.238,148.734
C02978=1160.279,212.256,-62.564,-177.860,7.236,148.735
C02979=1160.284,212.007,-62.539,-177.863,7.234,148.735
C02980=1160.288,211.758,-62.515,-177.866,7.231,148.735
C02981=1160.293,211.509,-62.490,-177.868,7.229,148.735
C02982=1160.298,211.261,-62.465,-177.871,7.226,148.735
C02983=1160.301,211.012,-62.440,-177.873,7.224,148.736
C02984=1160.306,210.763,-62.416,-177.877,7.221,148.736
C02985=1160.310,210.514,-62.391,-177.879,7.219,148.736
C02986=1160.315,210.244,-62.365,-177.882,7.217,148.736
C02987=1160.321,209.974,-62.338,-177.885,7.214,148.737
C02988=1160.325,209.703,-62.311,-177.888,7.211,148.737
C02989=1160.330,209.433,-62.284,-177.891,7.209,148.737
C02990=1160.335,209.183,-62.259,-177.893,7.207,148.737
C02991=1160.339,208.935,-62.235,-177.897,7.204,148.737
C02992=1160.344,208.686,-62.210,-177.899,7.202,148.738
C02993=1160.348,208.437,-62.186,-177.902,7.199,148.738
C02994=1160.353,208.188,-62.161,-177.904,7.197,148.738
C02995=1160.357,207.941,-62.136,-177.908,7.195,148.738
C02996=1160.362,207.691,-62.111,-177.910,7.192,148.738
C02997=1160.366,207.443,-62.087,-177.913,7.190,148.739
C02998=1160.371,207.194,-62.063,-177.915,7.188,148.739
C02999=1160.375,206.945,-62.038,-177.919,7.185,148.739
C03000=1160.380,206.696,-62.013,-177.921,7.183,148.740
C03001=1160.385,206.448,-61.989,-177.923,7.181,148.740
C03002=1160.390,206.199,-61.965,-177.927,7.179,148.740
C03003=1160.394,205.950,-61.940,-177.929,7.177,148.740
C03004=1160.399,205.701,-61.916,-177.932,7.174,148.740
C03005=1160.403,205.453,-61.892,-177.934,7.172,148.741
C03006=1160.408,205.204,-61.867,-177.938,7.169,148.741
C03007=1160.412,204.954,-61.843,-177.940,7.167,148.741
C03008=1160.417,204.706,-61.819,-177.943,7.165,148.741
C03009=1160.422,204.457,-61.794,-177.945,7.162,148.742
C03010=1160.426,204.208,-61.770,-177.949,7.160,148.742
C03011=1160.430,203.960,-61.746,-177.951,7.158,148.742
C03012=1160.435,203.711,-61.721,-177.954,7.155,148.742
C03013=1160.440,203.463,-61.697,-177.956,7.153,148.742
C03014=1160.444,203.214,-61.673,-177.959,7.150,148.743
C03015=1160.449,202.964,-61.649,-177.962,7.149,148.743
C03016=1160.453,202.716,-61.625,-177.965,7.146,148.743
C03017=1160.458,202.467,-61.601,-177.968,7.144,148.744
C03018=1160.463,202.219,-61.576,-177.970,7.141,148.744
C03019=1160.467,201.969,-61.552,-177.973,7.139,148.744
C03020=1160.471,201.720,-61.528,-177.975,7.137,148.744
C03021=1160.476,201.472,-61.504,-177.978,7.135,148.744
C03022=1160.481,201.223,-61.479,-177.981,7.133,148.745
C03023=1160.485,200.975,-61.455,-177.984,7.130,148.745
C03024=1160.489,200.725,-61.432,-177.987,7.128,148.745
C03025=1160.494,200.477,-61.408,-177.989,7.125,148.745
C03026=1160.499,200.228,-61.383,-177.992,7.123,148.746
C03027=1160.504,199.979,-61.360,-177.995,7.121,148.746
C03028=1160.508,199.731,-61.335,-177.998,7.119,148.746
C03029=1160.512,199.482,-61.311,-178.000,7.117,148.746
C03030=1160.517,199.232,-61.287,-178.003,7.114,148.747
C03031=1160.522,198.984,-61.263,-178.006,7.112,148.747
C03032=1160.526,198.735,-61.239,-178.008,7.109,148.747
C03033=1160.531,198.486,-61.216,-178.011,7.108,148.747
C03034=1160.535,198.238,-61.191,-178.014,7.105,148.748
C03035=1160.540,197.989,-61.168,-178.017,7.103,148.748
C03036=1160.545,197.740,-61.143,-178.019,7.101,148.748
C03037=1160.549,197.490,-61.120,-178.022,7.098,148.748
C03038=1160.553,197.242,-61.096,-178.025,7.096,148.749
C03039=1160.558,196.994,-61.072,-178.028,7.094,148.749
C03040=1160.562,196.744,-61.048,-178.030,7.092,148.749
C03041=1160.567,196.496,-61.024,-178.033,7.089,148.749
C03042=1160.572,196.247,-61.001,-178.036,7.087,148.750
C03043=1160.576,195.999,-60.977,-178.038,7.085,148.750
C03044=1160.581,195.749,-60.953,-178.042,7.083,148.750
C03045=1160.586,195.500,-60.929,-178.044,7.081,148.750
C03046=1160.590,195.252,-60.905,-178.047,7.078,148.751
C03047=1160.595,195.003,-60.882,-178.049,7.076,148.751
C03048=1160.600,194.754,-60.858,-178.052,7.074,148.751
C03049=1160.604,194.505,-60.835,-178.055,7.072,148.752
C03050=1160.608,194.256,-60.810,-178.057,7.070,148.752
C03051=1160.613,194.007,-60.787,-178.061,7.067,148.752
C03052=1160.617,193.758,-60.763,-178.063,7.065,148.752
C03053=1160.622,193.510,-60.739,-178.066,7.063,148.752
C03054=1160.627,193.261,-60.716,-178.069,7.060,148.753
C03055=1160.631,193.012,-60.693,-178.071,7.058,148.753
C03056=1160.636,192.763,-60.668,-178.074,7.056,148.753
C03057=1160.640,192.514,-60.645,-178.077,7.054,148.754
C03058=1160.645,192.265,-60.622,-178.079,7.052,148.754
C03059=1160.649,192.017,-60.598,-178.082,7.049,148.754
C03060=1160.654,191.768,-60.574,-178.085,7.048,148.754
C03061=1160.659,191.519,-60.551,-178.087,7.045,148.755
C03062=1160.664,191.270,-60.528,-178.091,7.043,148.755
C03063=1160.668,191.021,-60.504,-178.093,7.041,148.755
C03064=1160.673,190.772,-60.480,-178.096,7.038,148.755
C03065=1160.677,190.523,-60.457,-178.099,7.036,148.756
C03066=1160.682,190.274,-60.433,-178.101,7.035,148.756
C03067=1160.686,190.026,-60.409,-178.104,7.032,148.756
C03068=1160.692,189.777,-60.386,-178.107,7.030,148.757
C03069=1160.696,189.529,-60.364,-178.110,7.028,148.757
C03070=1160.700,189.280,-60.340,-178.112,7.025,148.757
C03071=1160.705,189.031,-60.317,-178.115,7.024,148.757
C03072=1160.710,188.782,-60.294,-178.118,7.022,148.758
C03073=1160.715,188.533,-60.270,-178.121,7.019,148.758
C03074=1160.719,188.284,-60.246,-178.123,7.017,148.758
C03075=1160.724,188.035,-60.223,-178.127,7.015,148.759
C03076=1160.728,187.786,-60.199,-178.129,7.012,148.759
C03077=1160.732,187.537,-60.177,-178.131,7.011,148.759
C03078=1160.737,187.288,-60.153,-178.135,7.008,148.759
C03079=1160.742,187.039,-60.130,-178.137,7.006,148.759
C03080=1160.746,186.790,-60.107,-178.140,7.004,148.760
C03081=1160.752,186.542,-60.084,-178.143,7.002,148.760
C03082=1160.756,186.293,-60.061,-178.145,7.000,148.761
C03083=1160.760,186.044,-60.037,-178.148,6.998,148.761
C03084=1160.765,185.795,-60.014,-178.151,6.995,148.761
C03085=1160.770,185.546,-59.991,-178.154,6.993,148.761
C03086=1160.774,185.297,-59.968,-178.156,6.991,148.762
C03087=1160.778,185.048,-59.945,-178.159,6.989,148.762
C03088=1160.783,184.799,-59.921,-178.162,6.987,148.762
C03089=1160.788,184.551,-59.898,-178.164,6.985,148.762
C03090=1160.793,184.282,-59.874,-178.167,6.982,148.763
C03091=1160.798,184.011,-59.848,-178.170,6.981,148.763
C03092=1160.803,183.741,-59.823,-178.173,6.978,148.763
C03093=1160.808,183.472,-59.799,-178.177,6.975,148.764
C03094=1160.813,183.224,-59.776,-178.179,6.974,148.764
C03095=1160.818,182.975,-59.753,-178.181,6.972,148.764
C03096=1160.822,182.726,-59.730,-178.185,6.969,148.765
C03097=1160.826,182.477,-59.706,-178.187,6.967,148.765
C03098=1160.831,182.228,-59.683,-178.190,6.966,148.765
C03099=1160.835,181.978,-59.661,-178.192,6.963,148.765
C03100=1160.841,181.730,-59.638,-178.196,6.961,148.766
C03101=1160.845,181.481,-59.615,-178.198,6.959,148.766
C03102=1160.849,181.232,-59.592,-178.200,6.957,148.766
C03103=1160.854,180.983,-59.569,-178.204,6.954,148.767
C03104=1160.858,180.734,-59.547,-178.206,6.953,148.767
C03105=1160.863,180.486,-59.524,-178.209,6.951,148.767
C03106=1160.868,180.237,-59.500,-178.212,6.948,148.767
C03107=1160.872,179.987,-59.478,-178.215,6.946,148.768
C03108=1160.877,179.738,-59.455,-178.217,6.944,148.768
C03109=1160.882,179.490,-59.432,-178.220,6.943,148.769
C03110=1160.886,179.241,-59.409,-178.223,6.940,148.769
C03111=1160.891,178.992,-59.386,-178.225,6.938,148.769
C03112=1160.895,178.743,-59.364,-178.228,6.936,148.769
C03113=1160.901,178.494,-59.341,-178.231,6.934,148.770
C03114=1160.905,178.245,-59.319,-178.234,6.932,148.770
C03115=1160.910,177.996,-59.295,-178.236,6.930,148.770
C03116=1160.914,177.747,-59.274,-178.239,6.928,148.771
C03117=1160.919,177.498,-59.250,-178.242,6.926,148.771
C03118=1160.923,177.250,-59.227,-178.245,6.924,148.771
C03119=1160.928,177.000,-59.205,-178.247,6.922,148.771
C03120=1160.933,176.752,-59.182,-178.250,6.919,148.772
C03121=1160.938,176.502,-59.160,-178.253,6.917,148.772
C03122=1160.942,176.254,-59.137,-178.256,6.916,148.772
C03123=1160.947,176.005,-59.115,-178.258,6.914,148.773
C03124=1160.951,175.756,-59.092,-178.261,6.911,148.773
C03125=1160.956,175.507,-59.070,-178.264,6.909,148.773
C03126=1160.961,175.258,-59.047,-178.267,6.907,148.774
C03127=1160.965,175.009,-59.025,-178.269,6.906,148.774
C03128=1160.970,174.760,-59.001,-178.272,6.903,148.774
C03129=1160.975,174.511,-58.980,-178.275,6.901,148.775
C03130=1160.979,174.262,-58.956,-178.277,6.899,148.775
C03131=1160.984,174.013,-58.934,-178.280,6.898,148.775
C03132=1160.988,173.765,-58.912,-178.283,6.895,148.776
C03133=1160.993,173.515,-58.889,-178.286,6.893,148.776
C03134=1160.997,173.266,-58.867,-178.288,6.891,148.776
C03135=1161.002,173.018,-58.845,-178.291,6.889,148.777
C03136=1161.007,172.768,-58.822,-178.294,6.887,148.777
C03137=1161.012,172.520,-58.801,-178.297,6.885,148.777
C03138=1161.017,172.271,-58.777,-178.299,6.883,148.777
C03139=1161.021,172.021,-58.755,-178.302,6.881,148.778
C03140=1161.026,171.773,-58.733,-178.305,6.879,148.778
C03141=1161.030,171.524,-58.710,-178.308,6.877,148.778
C03142=1161.035,171.275,-58.688,-178.311,6.875,148.779
C03143=1161.040,171.026,-58.666,-178.313,6.873,148.779
C03144=1161.044,170.778,-58.644,-178.315,6.871,148.779
C03145=1161.049,170.528,-58.621,-178.319,6.869,148.780
C03146=1161.053,170.279,-58.599,-178.321,6.867,148.780
C03147=1161.058,170.030,-58.578,-178.324,6.865,148.780
C03148=1161.063,169.781,-58.554,-178.327,6.863,148.781
C03149=1161.068,169.532,-58.533,-178.330,6.861,148.781
C03150=1161.072,169.283,-58.511,-178.332,6.859,148.781
C03151=1161.077,169.034,-58.489,-178.335,6.857,148.782
C03152=1161.082,168.785,-58.466,-178.338,6.855,148.782
C03153=1161.087,168.537,-58.444,-178.340,6.854,148.782
C03154=1161.091,168.287,-58.422,-178.344,6.851,148.783
C03155=1161.096,168.039,-58.400,-178.346,6.849,148.783
C03156=1161.101,167.789,-58.377,-178.349,6.847,148.783
C03157=1161.106,167.540,-58.356,-178.351,6.845,148.784
C03158=1161.110,167.291,-58.334,-178.354,6.844,148.784
C03159=1161.115,167.042,-58.312,-178.357,6.841,148.784
C03160=1161.119,166.794,-58.289,-178.360,6.839,148.785
C03161=1161.124,166.545,-58.268,-178.363,6.838,148.785
C03162=1161.129,166.295,-58.245,-178.365,6.836,148.785
C03163=1161.133,166.047,-58.223,-178.367,6.834,148.786
C03164=1161.138,165.797,-58.201,-178.371,6.831,148.786
C03165=1161.143,165.549,-58.180,-178.373,6.829,148.786
C03166=1161.147,165.299,-58.157,-178.376,6.828,148.787
C03167=1161.152,165.051,-58.136,-178.379,6.826,148.787
C03168=1161.156,164.801,-58.114,-178.382,6.824,148.787
C03169=1161.161,164.553,-58.092,-178.384,6.822,148.788
C03170=1161.166,164.303,-58.069,-178.387,6.820,148.788
C03171=1161.171,164.054,-58.048,-178.390,6.818,148.788
C03172=1161.175,163.805,-58.026,-178.392,6.816,148.789
C03173=1161.180,163.556,-58.004,-178.395,6.814,148.789
C03174=1161.185,163.308,-57.982,-178.398,6.813,148.789
C03175=1161.189,163.058,-57.960,-178.400,6.811,148.790
C03176=1161.194,162.810,-57.939,-178.404,6.808,148.790
C03177=1161.198,162.560,-57.917,-178.406,6.806,148.790
C03178=1161.203,162.311,-57.896,-178.409,6.804,148.791
C03179=1161.208,162.062,-57.874,-178.411,6.803,148.791
C03180=1161.212,161.813,-57.852,-178.414,6.801,148.791
C03181=1161.217,161.565,-57.830,-178.417,6.799,148.792
C03182=1161.222,161.315,-57.808,-178.420,6.797,148.792
C03183=1161.226,161.067,-57.786,-178.423,6.795,148.793
C03184=1161.231,160.817,-57.765,-178.425,6.793,148.793
C03185=1161.236,160.568,-57.743,-178.428,6.791,148.793
C03186=1161.241,160.319,-57.722,-178.431,6.790,148.794
C03187=1161.245,160.070,-57.700,-178.433,6.788,148.794
C03188=1161.250,159.821,-57.678,-178.436,6.786,148.794
C03189=1161.255,159.572,-57.657,-178.439,6.783,148.795
C03190=1161.259,159.323,-57.635,-178.442,6.782,148.795
C03191=1161.264,159.074,-57.613,-178.444,6.780,148.795
C03192=1161.269,158.826,-57.592,-178.447,6.778,148.796
C03193=1161.274,158.576,-57.570,-178.450,6.776,148.796
C03194=1161.278,158.307,-57.547,-178.453,6.774,148.796
C03195=1161.284,158.038,-57.523,-178.456,6.772,148.797
C03196=1161.288,157.769,-57.501,-178.458,6.770,148.797
C03197=1161.294,157.500,-57.478,-178.462,6.768,148.798
C03198=1161.298,157.251,-57.456,-178.464,6.766,148.798
C03199=1161.303,157.002,-57.435,-178.467,6.764,148.798
C03200=1161.308,156.753,-57.414,-178.470,6.763,148.799
C03201=1161.312,156.504,-57.392,-178.473,6.761,148.799
C03202=1161.317,156.255,-57.370,-178.475,6.759,148.799
C03203=1161.322,156.006,-57.349,-178.478,6.757,148.800
C03204=1161.326,155.758,-57.328,-178.481,6.756,148.800
C03205=1161.331,155.508,-57.306,-178.484,6.753,148.801
C03206=1161.336,155.259,-57.285,-178.487,6.751,148.801
C03207=1161.341,155.010,-57.264,-178.489,6.750,148.801
C03208=1161.345,154.760,-57.242,-178.492,6.747,148.801
C03209=1161.350,154.512,-57.220,-178.494,6.746,148.802
C03210=1161.355,154.263,-57.200,-178.497,6.744,148.802
C03211=1161.359,154.014,-57.178,-178.500,6.742,148.803
C03212=1161.364,153.764,-57.157,-178.502,6.740,148.803
C03213=1161.369,153.516,-57.135,-178.505,6.739,148.803
C03214=1161.373,153.267,-57.115,-178.508,6.736,148.804
C03215=1161.379,153.017,-57.094,-178.511,6.734,148.804
C03216=1161.383,152.769,-57.072,-178.514,6.733,148.804
C03217=1161.388,152.519,-57.051,-178.516,6.731,148.805
C03218=1161.392,152.270,-57.030,-178.519,6.729,148.805
C03219=1161.397,152.021,-57.009,-178.522,6.727,148.806
C03220=1161.402,151.773,-56.987,-178.524,6.726,148.806
C03221=1161.407,151.523,-56.966,-178.527,6.724,148.806
C03222=1161.411,151.274,-56.945,-178.530,6.722,148.807
C03223=1161.416,151.025,-56.924,-178.533,6.721,148.807
C03224=1161.421,150.776,-56.903,-178.535,6.719,148.808
C03225=1161.426,150.527,-56.882,-178.538,6.717,148.808
C03226=1161.430,150.278,-56.861,-178.541,6.715,148.808
C03227=1161.436,150.029,-56.840,-178.544,6.713,148.809
C03228=1161.440,149.779,-56.819,-178.547,6.711,148.809
C03229=1161.444,149.531,-56.797,-178.549,6.709,148.809
C03230=1161.450,149.281,-56.776,-178.552,6.708,148.810
C03231=1161.454,149.032,-56.756,-178.555,6.706,148.810
C03232=1161.459,148.784,-56.734,-178.557,6.704,148.811
C03233=1161.463,148.535,-56.714,-178.560,6.702,148.811
C03234=1161.468,148.285,-56.692,-178.563,6.701,148.811
C03235=1161.473,148.036,-56.671,-178.566,6.699,148.812
C03236=1161.477,147.787,-56.650,-178.568,6.697,148.812
C03237=1161.482,147.538,-56.629,-178.571,6.695,148.812
C03238=1161.487,147.289,-56.609,-178.574,6.694,148.813
C03239=1161.492,147.040,-56.588,-178.576,6.692,148.813
C03240=1161.496,146.791,-56.568,-178.579,6.690,148.814
C03241=1161.502,146.542,-56.547,-178.582,6.688,148.814
C03242=1161.506,146.293,-56.525,-178.584,6.687,148.814
C03243=1161.511,146.044,-56.505,-178.587,6.685,148.815
C03244=1161.515,145.794,-56.483,-178.590,6.682,148.815
C03245=1161.520,145.545,-56.463,-178.593,6.681,148.816
C03246=1161.525,145.296,-56.442,-178.596,6.679,148.816
C03247=1161.530,145.047,-56.422,-178.599,6.677,148.816
C03248=1161.535,144.798,-56.401,-178.601,6.676,148.817
C03249=1161.539,144.549,-56.380,-178.604,6.674,148.817
C03250=1161.544,144.300,-56.359,-178.607,6.672,148.817
C03251=1161.548,144.051,-56.338,-178.609,6.670,148.818
C03252=1161.554,143.802,-56.317,-178.612,6.669,148.818
C03253=1161.558,143.553,-56.297,-178.615,6.667,148.819
C03254=1161.562,143.304,-56.277,-178.618,6.665,148.819
C03255=1161.568,143.055,-56.256,-178.620,6.663,148.819
C03256=1161.572,142.806,-56.235,-178.623,6.662,148.820
C03257=1161.577,142.556,-56.214,-178.626,6.660,148.820
C03258=1161.582,142.307,-56.194,-178.628,6.658,148.821
C03259=1161.587,142.058,-56.173,-178.631,6.656,148.821
C03260=1161.591,141.809,-56.152,-178.634,6.655,148.821
C03261=1161.596,141.560,-56.132,-178.636,6.653,148.822
C03262=1161.601,141.311,-56.111,-178.639,6.651,148.822
C03263=1161.606,141.061,-56.091,-178.642,6.650,148.822
C03264=1161.610,140.813,-56.071,-178.645,6.648,148.823
C03265=1161.615,140.563,-56.050,-178.647,6.646,148.823
C03266=1161.620,140.314,-56.030,-178.650,6.644,148.824
C03267=1161.625,140.065,-56.009,-178.653,6.643,148.824
C03268=1161.629,139.816,-55.988,-178.655,6.641,148.824
C03269=1161.634,139.567,-55.968,-178.658,6.639,148.825
C03270=1161.639,139.318,-55.947,-178.661,6.637,148.825
C03271=1161.644,139.068,-55.927,-178.663,6.636,148.826
C03272=1161.648,138.819,-55.907,-178.666,6.634,148.826
C03273=1161.653,138.570,-55.887,-178.669,6.632,148.826
C03274=1161.658,138.321,-55.866,-178.672,6.631,148.827
C03275=1161.662,138.072,-55.845,-178.675,6.629,148.827
C03276=1161.667,137.823,-55.826,-178.677,6.627,148.828
C03277=1161.672,137.573,-55.805,-178.680,6.626,148.828
C03278=1161.677,137.324,-55.784,-178.683,6.624,148.828
C03279=1161.681,137.075,-55.764,-178.686,6.622,148.829
C03280=1161.686,136.826,-55.744,-178.688,6.621,148.829
C03281=1161.691,136.577,-55.724,-178.691,6.619,148.830
C03282=1161.696,136.328,-55.703,-178.694,6.617,148.830
C03283=1161.700,136.079,-55.683,-178.696,6.615,148.830
C03284=1161.705,135.830,-55.663,-178.699,6.614,148.831
C03285=1161.710,135.581,-55.642,-178.702,6.612,148.831
C03286=1161.715,135.332,-55.622,-178.705,6.610,148.832
C03287=1161.719,135.082,-55.602,-178.707,6.608,148.832
C03288=1161.724,134.833,-55.582,-178.710,6.607,148.833
C03289=1161.728,134.584,-55.562,-178.713,6.606,148.833
C03290=1161.734,134.335,-55.542,-178.715,6.604,148.833
C03291=1161.739,134.086,-55.521,-178.718,6.603,148.834
C03292=1161.744,133.837,-55.502,-178.721,6.601,148.834
C03293=1161.748,133.588,-55.481,-178.723,6.599,148.835
C03294=1161.752,133.339,-55.461,-178.726,6.598,148.835
C03295=1161.757,133.089,-55.441,-178.729,6.596,148.835
C03296=1161.762,132.841,-55.421,-178.732,6.594,148.836
C03297=1161.768,132.591,-55.401,-178.734,6.592,148.836
C03298=1161.772,132.323,-55.379,-178.737,6.591,148.837
C03299=1161.778,132.054,-55.358,-178.740,6.589,148.837
C03300=1161.783,131.785,-55.336,-178.743,6.587,148.838
C03301=1161.788,131.517,-55.315,-178.746,6.585,148.838
C03302=1161.793,131.267,-55.294,-178.749,6.583,148.838
C03303=1161.797,131.018,-55.274,-178.752,6.582,148.839
C03304=1161.802,130.769,-55.254,-178.755,6.580,148.839
C03305=1161.807,130.521,-55.234,-178.757,6.579,148.840
C03306=1161.812,130.271,-55.215,-178.760,6.578,148.840
C03307=1161.817,130.021,-55.195,-178.762,6.576,148.841
C03308=1161.821,129.773,-55.175,-178.765,6.574,148.841
C03309=1161.826,129.523,-55.155,-178.768,6.572,148.841
C03310=1161.831,129.275,-55.135,-178.770,6.571,148.842
C03311=1161.836,129.025,-55.115,-178.773,6.569,148.842
C03312=1161.840,128.776,-55.095,-178.776,6.568,148.843
C03313=1161.845,128.527,-55.075,-178.779,6.566,148.843
C03314=1161.850,128.278,-55.056,-178.782,6.564,148.844
C03315=1161.855,128.029,-55.036,-178.784,6.562,148.844
C03316=1161.859,127.779,-55.016,-178.787,6.561,148.844
C03317=1161.864,127.530,-54.996,-178.789,6.560,148.845
C03318=1161.869,127.281,-54.976,-178.792,6.558,148.845
C03319=1161.874,127.032,-54.957,-178.795,6.556,148.846
C03320=1161.879,126.782,-54.937,-178.798,6.555,148.846
C03321=1161.884,126.533,-54.918,-178.801,6.553,148.847
C03322=1161.888,126.284,-54.897,-178.803,6.552,148.847
C03323=1161.893,126.035,-54.878,-178.806,6.550,148.847
C03324=1161.898,125.785,-54.858,-178.809,6.548,148.848
C03325=1161.903,125.537,-54.838,-178.811,6.546,148.848
C03326=1161.907,125.288,-54.819,-178.814,6.545,148.849
C03327=1161.912,125.038,-54.799,-178.817,6.544,148.849
C03328=1161.917,124.789,-54.780,-178.819,6.542,148.850
C03329=1161.922,124.540,-54.760,-178.822,6.541,148.850
C03330=1161.926,124.291,-54.740,-178.825,6.539,148.850
C03331=1161.932,124.042,-54.721,-178.828,6.537,148.851
C03332=1161.936,123.792,-54.701,-178.830,6.535,148.851
C03333=1161.941,123.543,-54.681,-178.833,6.534,148.852
C03334=1161.946,123.294,-54.663,-178.836,6.532,148.852
C03335=1161.950,123.045,-54.643,-178.839,6.531,148.853
C03336=1161.955,122.796,-54.623,-178.841,6.530,148.853
C03337=1161.960,122.547,-54.603,-178.844,6.528,148.853
C03338=1161.965,122.297,-54.584,-178.847,6.526,148.854
C03339=1161.970,122.048,-54.564,-178.849,6.525,148.854
C03340=1161.974,121.799,-54.545,-178.852,6.523,148.855
C03341=1161.979,121.550,-54.526,-178.855,6.522,148.855
C03342=1161.984,121.301,-54.506,-178.858,6.520,148.856
C03343=1161.989,121.051,-54.487,-178.860,6.519,148.856
C03344=1161.994,120.802,-54.467,-178.863,6.517,148.856
C03345=1161.998,120.553,-54.448,-178.865,6.515,148.857
C03346=1162.003,120.304,-54.429,-178.869,6.514,148.857
C03347=1162.009,120.055,-54.410,-178.871,6.512,148.858
C03348=1162.013,119.805,-54.390,-178.874,6.511,148.858
C03349=1162.017,119.556,-54.371,-178.877,6.509,148.859
C03350=1162.023,119.307,-54.352,-178.879,6.508,148.859
C03351=1162.027,119.057,-54.332,-178.882,6.506,148.859
C03352=1162.033,118.809,-54.313,-178.885,6.505,148.860
C03353=1162.037,118.559,-54.293,-178.887,6.503,148.860
C03354=1162.042,118.310,-54.274,-178.890,6.502,148.861
C03355=1162.047,118.061,-54.255,-178.893,6.500,148.861
C03356=1162.051,117.812,-54.235,-178.896,6.498,148.862
C03357=1162.056,117.563,-54.216,-178.898,6.497,148.862
C03358=1162.061,117.313,-54.197,-178.901,6.496,148.863
C03359=1162.066,117.064,-54.179,-178.904,6.494,148.863
C03360=1162.071,116.814,-54.159,-178.906,6.492,148.863
C03361=1162.076,116.566,-54.140,-178.909,6.491,148.864
C03362=1162.080,116.316,-54.121,-178.912,6.489,148.864
C03363=1162.085,116.067,-54.101,-178.914,6.488,148.865
C03364=1162.090,115.818,-54.082,-178.917,6.487,148.865
C03365=1162.095,115.569,-54.063,-178.920,6.485,148.866
C03366=1162.100,115.319,-54.044,-178.923,6.483,148.866
C03367=1162.105,115.070,-54.025,-178.925,6.482,148.867
C03368=1162.109,114.821,-54.006,-178.928,6.481,148.867
C03369=1162.114,114.572,-53.986,-178.931,6.479,148.868
C03370=1162.119,114.322,-53.968,-178.933,6.478,148.868
C03371=1162.124,114.073,-53.949,-178.936,6.476,148.868
C03372=1162.129,113.824,-53.929,-178.939,6.474,148.869
C03373=1162.133,113.575,-53.910,-178.941,6.474,148.869
C03374=1162.138,113.325,-53.891,-178.944,6.472,148.870
C03375=1162.143,113.077,-53.873,-178.947,6.470,148.870
C03376=1162.148,112.827,-53.853,-178.950,6.469,148.871
C03377=1162.152,112.578,-53.834,-178.953,6.467,148.871
C03378=1162.158,112.329,-53.816,-178.955,6.465,148.872
C03379=1162.162,112.080,-53.797,-178.958,6.465,148.872
C03380=1162.167,111.831,-53.777,-178.960,6.463,148.873
C03381=1162.172,111.581,-53.759,-178.963,6.461,148.873
C03382=1162.177,111.332,-53.740,-178.966,6.460,148.874
C03383=1162.181,111.082,-53.721,-178.968,6.459,148.874
C03384=1162.187,110.833,-53.702,-178.971,6.457,148.874
C03385=1162.191,110.585,-53.683,-178.974,6.456,148.875
C03386=1162.196,110.335,-53.665,-178.977,6.454,148.875
C03387=1162.201,110.086,-53.646,-178.980,6.452,148.876
C03388=1162.206,109.836,-53.627,-178.982,6.452,148.876
C03389=1162.211,109.587,-53.608,-178.985,6.450,148.877
C03390=1162.216,109.338,-53.589,-178.987,6.448,148.877
C03391=1162.220,109.089,-53.571,-178.990,6.447,148.878
C03392=1162.226,108.840,-53.551,-178.993,6.445,148.878
C03393=1162.230,108.590,-53.533,-178.995,6.444,148.878
C03394=1162.234,108.341,-53.514,-178.998,6.442,148.879
C03395=1162.240,108.092,-53.496,-179.001,6.441,148.880
C03396=1162.244,107.842,-53.477,-179.004,6.439,148.880
C03397=1162.250,107.593,-53.458,-179.006,6.439,148.880
C03398=1162.254,107.344,-53.439,-179.009,6.437,148.881
C03399=1162.259,107.095,-53.421,-179.012,6.435,148.881
C03400=1162.264,106.845,-53.402,-179.015,6.434,148.882
C03401=1162.269,106.597,-53.384,-179.017,6.433,148.882
C03402=1162.274,106.327,-53.363,-179.020,6.431,148.883
C03403=1162.279,106.060,-53.343,-179.023,6.430,148.883
C03404=1162.285,105.791,-53.323,-179.026,6.428,148.884
C03405=1162.290,105.523,-53.304,-179.029,6.427,148.884
C03406=1162.295,105.273,-53.284,-179.031,6.425,148.885
C03407=1162.300,105.024,-53.266,-179.034,6.423,148.885
C03408=1162.304,104.775,-53.248,-179.037,6.422,148.886
C03409=1162.309,104.525,-53.229,-179.040,6.421,148.886
C03410=1162.314,104.276,-53.211,-179.042,6.419,148.887
C03411=1162.319,104.027,-53.193,-179.045,6.418,148.887
C03412=1162.323,103.778,-53.173,-179.048,6.417,148.888
C03413=1162.329,103.528,-53.155,-179.050,6.415,148.888
C03414=1162.334,103.279,-53.137,-179.053,6.414,148.888
C03415=1162.338,103.030,-53.118,-179.056,6.412,148.889
C03416=1162.342,102.781,-53.100,-179.058,6.411,148.890
C03417=1162.348,102.531,-53.081,-179.061,6.410,148.890
C03418=1162.353,102.282,-53.063,-179.064,6.408,148.890
C03419=1162.358,102.033,-53.045,-179.067,6.406,148.891
C03420=1162.362,101.783,-53.026,-179.069,6.406,148.891
C03421=1162.368,101.534,-53.008,-179.072,6.404,148.892
C03422=1162.373,101.285,-52.990,-179.075,6.402,148.892
C03423=1162.377,101.036,-52.972,-179.077,6.402,148.893
C03424=1162.381,100.786,-52.953,-179.080,6.400,148.893
C03425=1162.387,100.537,-52.934,-179.083,6.398,148.894
C03426=1162.392,100.288,-52.916,-179.085,6.397,148.894
C03427=1162.397,100.039,-52.898,-179.088,6.396,148.895
C03428=1162.402,99.789,-52.880,-179.091,6.395,148.895
C03429=1162.406,99.540,-52.861,-179.093,6.393,148.896
C03430=1162.411,99.291,-52.843,-179.096,6.392,148.896
C03431=1162.416,99.041,-52.825,-179.099,6.391,148.897
C03432=1162.421,98.792,-52.807,-179.101,6.389,148.897
C03433=1162.426,98.542,-52.788,-179.104,6.387,148.897
C03434=1162.431,98.293,-52.770,-179.107,6.387,148.898
C03435=1162.435,98.044,-52.752,-179.110,6.385,148.899
C03436=1162.440,97.795,-52.734,-179.112,6.383,148.899
C03437=1162.445,97.546,-52.716,-179.115,6.383,148.900
C03438=1162.450,97.297,-52.698,-179.118,6.381,148.900
C03439=1162.455,97.046,-52.679,-179.120,6.379,148.900
C03440=1162.460,96.797,-52.661,-179.122,6.378,148.901
C03441=1162.465,96.548,-52.643,-179.126,6.377,148.901
C03442=1162.470,96.299,-52.625,-179.128,6.375,148.902
C03443=1162.475,96.050,-52.607,-179.131,6.374,148.902
C03444=1162.479,95.801,-52.589,-179.134,6.373,148.903
C03445=1162.485,95.551,-52.572,-179.136,6.371,148.903
C03446=1162.489,95.301,-52.553,-179.139,6.370,148.904
C03447=1162.494,95.052,-52.535,-179.142,6.369,148.904
C03448=1162.499,94.803,-52.517,-179.145,6.368,148.905
C03449=1162.504,94.554,-52.499,-179.147,6.366,148.905
C03450=1162.509,94.305,-52.481,-179.150,6.365,148.906
C03451=1162.514,94.056,-52.463,-179.153,6.364,148.906
C03452=1162.518,93.806,-52.445,-179.155,6.362,148.907
C03453=1162.523,93.557,-52.427,-179.158,6.361,148.907
C03454=1162.528,93.308,-52.409,-179.161,6.360,148.908
C03455=1162.533,93.058,-52.391,-179.163,6.358,148.908
C03456=1162.538,92.809,-52.373,-179.166,6.357,148.909
C03457=1162.543,92.559,-52.356,-179.169,6.356,148.909
C03458=1162.548,92.310,-52.338,-179.172,6.354,148.910
C03459=1162.553,92.061,-52.320,-179.174,6.353,148.910
C03460=1162.557,91.812,-52.302,-179.177,6.352,148.911
C03461=1162.562,91.562,-52.284,-179.180,6.350,148.911
C03462=1162.567,91.313,-52.266,-179.182,6.349,148.912
C03463=1162.573,91.063,-52.249,-179.185,6.348,148.912
C03464=1162.577,90.814,-52.231,-179.188,6.346,148.913
C03465=1162.582,90.565,-52.213,-179.190,6.345,148.913
C03466=1162.587,90.316,-52.195,-179.193,6.344,148.914
C03467=1162.591,90.067,-52.177,-179.195,6.343,148.914
C03468=1162.597,89.817,-52.160,-179.198,6.341,148.915
C03469=1162.602,89.568,-52.142,-179.201,6.340,148.915
C03470=1162.606,89.319,-52.124,-179.203,6.339,148.916
C03471=1162.612,89.069,-52.107,-179.206,6.338,148.916
C03472=1162.617,88.820,-52.089,-179.209,6.336,148.917
C03473=1162.621,88.571,-52.071,-179.211,6.335,148.917
C03474=1162.626,88.322,-52.053,-179.214,6.334,148.918
C03475=1162.631,88.072,-52.036,-179.217,6.332,148.918
C03476=1162.636,87.823,-52.018,-179.219,6.331,148.919
C03477=1162.641,87.574,-52.000,-179.222,6.330,148.919
C03478=1162.646,87.324,-51.983,-179.225,6.329,148.920
C03479=1162.651,87.075,-51.965,-179.227,6.328,148.920
C03480=1162.655,86.825,-51.948,-179.230,6.326,148.921
C03481=1162.660,86.576,-51.930,-179.233,6.325,148.921
C03482=1162.665,86.327,-51.912,-179.236,6.324,148.922
C03483=1162.670,86.077,-51.895,-179.238,6.323,148.922
C03484=1162.675,85.828,-51.877,-179.241,6.321,148.923
C03485=1162.680,85.579,-51.860,-179.244,6.320,148.923
C03486=1162.685,85.329,-51.842,-179.246,6.319,148.924
C03487=1162.690,85.080,-51.824,-179.249,6.317,148.924
C03488=1162.695,84.830,-51.807,-179.252,6.316,148.925
C03489=1162.699,84.582,-51.790,-179.254,6.315,148.925
C03490=1162.704,84.332,-51.773,-179.257,6.314,148.926
C03491=1162.709,84.083,-51.755,-179.259,6.313,148.926
C03492=1162.714,83.833,-51.737,-179.262,6.311,148.927
C03493=1162.718,83.584,-51.720,-179.265,6.310,148.927
C03494=1162.724,83.334,-51.703,-179.267,6.309,148.928
C03495=1162.729,83.085,-51.685,-179.271,6.307,148.928
C03496=1162.734,82.836,-51.668,-179.273,6.307,148.929
C03497=1162.739,82.587,-51.650,-179.275,6.305,148.929
C03498=1162.744,82.337,-51.633,-179.279,6.304,148.930
C03499=1162.749,82.088,-51.615,-179.281,6.303,148.930
C03500=1162.753,81.839,-51.598,-179.284,6.301,148.931
C03501=1162.758,81.589,-51.581,-179.286,6.300,148.931
C03502=1162.763,81.340,-51.563,-179.289,6.299,148.932
C03503=1162.768,81.090,-51.547,-179.291,6.298,148.932
C03504=1162.773,80.841,-51.529,-179.294,6.297,148.933
C03505=1162.779,80.592,-51.512,-179.297,6.295,148.933
C03506=1162.783,80.323,-51.494,-179.300,6.294,148.934
C03507=1162.789,80.054,-51.475,-179.303,6.293,148.934
C03508=1162.794,79.787,-51.456,-179.306,6.291,148.935
C03509=1162.799,79.518,-51.438,-179.309,6.290,148.936
C03510=1162.804,79.268,-51.420,-179.311,6.289,148.936
C03511=1162.809,79.019,-51.403,-179.314,6.287,148.936
C03512=1162.814,78.770,-51.386,-179.316,6.287,148.937
C03513=1162.819,78.521,-51.369,-179.319,6.285,148.937
C03514=1162.824,78.271,-51.352,-179.322,6.284,148.938
C03515=1162.829,78.022,-51.334,-179.324,6.283,148.939
C03516=1162.833,77.773,-51.318,-179.327,6.281,148.939
C03517=1162.838,77.523,-51.300,-179.330,6.281,148.940
C03518=1162.844,77.274,-51.283,-179.332,6.279,148.940
C03519=1162.848,77.025,-51.266,-179.335,6.278,148.941
C03520=1162.854,76.775,-51.249,-179.338,6.277,148.941
C03521=1162.858,76.526,-51.232,-179.340,6.276,148.942
C03522=1162.863,76.276,-51.215,-179.343,6.275,148.942
C03523=1162.868,76.028,-51.198,-179.346,6.273,148.943
C03524=1162.873,75.778,-51.181,-179.348,6.272,148.943
C03525=1162.878,75.528,-51.164,-179.351,6.271,148.944
C03526=1162.883,75.278,-51.147,-179.353,6.270,148.944
C03527=1162.888,75.029,-51.130,-179.357,6.269,148.945
C03528=1162.893,74.780,-51.113,-179.359,6.268,148.945
C03529=1162.898,74.531,-51.096,-179.361,6.266,148.946
C03530=1162.903,74.281,-51.078,-179.364,6.266,148.946
C03531=1162.907,74.032,-51.062,-179.367,6.264,148.947
C03532=1162.912,73.783,-51.045,-179.369,6.263,148.947
C03533=1162.918,73.533,-51.028,-179.372,6.262,148.948
C03534=1162.922,73.284,-51.012,-179.374,6.261,148.948
C03535=1162.927,73.034,-50.994,-179.378,6.260,148.949
C03536=1162.932,72.785,-50.978,-179.380,6.259,148.949
C03537=1162.938,72.535,-50.961,-179.383,6.257,148.950
C03538=1162.942,72.286,-50.944,-179.386,6.256,148.950
C03539=1162.947,72.037,-50.928,-179.388,6.255,148.951
C03540=1162.952,71.787,-50.910,-179.391,6.253,148.952
C03541=1162.957,71.538,-50.894,-179.393,6.253,148.952
C03542=1162.962,71.288,-50.877,-179.396,6.251,148.953
C03543=1162.967,71.039,-50.860,-179.399,6.250,148.953
C03544=1162.972,70.790,-50.844,-179.402,6.249,148.954
C03545=1162.977,70.540,-50.826,-179.404,6.248,148.954
C03546=1162.982,70.291,-50.810,-179.407,6.247,148.955
C03547=1162.986,70.042,-50.793,-179.409,6.246,148.955
C03548=1162.992,69.792,-50.776,-179.412,6.244,148.956
C03549=1162.997,69.543,-50.760,-179.415,6.244,148.956
C03550=1163.001,69.294,-50.743,-179.417,6.242,148.957
C03551=1163.006,69.044,-50.726,-179.420,6.241,148.957
C03552=1163.011,68.795,-50.710,-179.423,6.240,148.958
C03553=1163.016,68.546,-50.693,-179.425,6.239,148.958
C03554=1163.021,68.296,-50.676,-179.428,6.238,148.959
C03555=1163.026,68.047,-50.659,-179.430,6.237,148.959
C03556=1163.031,67.797,-50.643,-179.434,6.236,148.960
C03557=1163.036,67.547,-50.626,-179.436,6.235,148.960
C03558=1163.041,67.298,-50.610,-179.438,6.233,148.961
C03559=1163.046,67.049,-50.593,-179.441,6.233,148.962
C03560=1163.051,66.800,-50.577,-179.444,6.231,148.962
C03561=1163.056,66.550,-50.560,-179.446,6.230,148.963
C03562=1163.061,66.301,-50.543,-179.449,6.229,148.963
C03563=1163.066,66.052,-50.527,-179.452,6.228,148.964
C03564=1163.070,65.802,-50.511,-179.455,6.227,148.964
C03565=1163.076,65.553,-50.494,-179.457,6.226,148.965
C03566=1163.081,65.303,-50.477,-179.459,6.225,148.965
C03567=1163.085,65.054,-50.460,-179.462,6.223,148.966
C03568=1163.091,64.804,-50.445,-179.465,6.223,148.966
C03569=1163.095,64.555,-50.428,-179.467,6.221,148.967
C03570=1163.101,64.306,-50.411,-179.470,6.221,148.967
C03571=1163.105,64.056,-50.395,-179.473,6.219,148.968
C03572=1163.110,63.806,-50.379,-179.475,6.218,148.968
C03573=1163.115,63.557,-50.362,-179.478,6.217,148.969
C03574=1163.120,63.308,-50.346,-179.480,6.216,148.969
C03575=1163.125,63.059,-50.330,-179.484,6.215,148.970
C03576=1163.130,62.809,-50.313,-179.486,6.214,148.971
C03577=1163.135,62.560,-50.296,-179.489,6.213,148.971
C03578=1163.140,62.310,-50.280,-179.491,6.212,148.972
C03579=1163.145,62.061,-50.264,-179.494,6.210,148.972
C03580=1163.150,61.812,-50.248,-179.496,6.210,148.973
C03581=1163.155,61.561,-50.232,-179.499,6.209,148.973
C03582=1163.160,61.313,-50.215,-179.502,6.207,148.974
C03583=1163.165,61.063,-50.198,-179.504,6.206,148.974
C03584=1163.170,60.813,-50.182,-179.507,6.205,148.975
C03585=1163.175,60.564,-50.166,-179.509,6.204,148.975
C03586=1163.180,60.315,-50.150,-179.513,6.203,148.976
C03587=1163.185,60.065,-50.134,-179.515,6.202,148.976
C03588=1163.190,59.816,-50.117,-179.518,6.201,148.977
C03589=1163.194,59.566,-50.101,-179.520,6.200,148.978
C03590=1163.200,59.317,-50.085,-179.523,6.199,148.978
C03591=1163.204,59.067,-50.069,-179.525,6.198,148.979
C03592=1163.209,58.819,-50.053,-179.528,6.197,148.979
C03593=1163.214,58.568,-50.037,-179.531,6.196,148.980
C03594=1163.219,58.320,-50.020,-179.533,6.195,148.980
C03595=1163.225,58.070,-50.005,-179.536,6.193,148.981
C03596=1163.229,57.821,-49.988,-179.538,6.193,148.981
C03597=1163.234,57.571,-49.973,-179.541,6.192,148.982
C03598=1163.239,57.322,-49.956,-179.544,6.190,148.982
C03599=1163.244,57.073,-49.940,-179.546,6.190,148.983
C03600=1163.249,56.823,-49.924,-179.549,6.188,148.984
C03601=1163.254,56.574,-49.908,-179.552,6.188,148.984
C03602=1163.259,56.324,-49.891,-179.554,6.186,148.985
C03603=1163.264,56.075,-49.876,-179.557,6.186,148.985
C03604=1163.269,55.825,-49.860,-179.559,6.185,148.986
C03605=1163.274,55.576,-49.844,-179.562,6.183,148.986
C03606=1163.279,55.326,-49.828,-179.565,6.183,148.987
C03607=1163.284,55.077,-49.811,-179.567,6.181,148.987
C03608=1163.289,54.828,-49.796,-179.570,6.180,148.988
C03609=1163.294,54.577,-49.780,-179.572,6.180,148.988
C03610=1163.299,54.310,-49.762,-179.575,6.178,148.989
C03611=1163.305,54.041,-49.745,-179.579,6.177,148.990
C03612=1163.310,53.773,-49.728,-179.581,6.176,148.990
C03613=1163.316,53.504,-49.711,-179.584,6.175,148.991
C03614=1163.321,53.254,-49.695,-179.586,6.174,148.991
C03615=1163.326,53.005,-49.679,-179.589,6.173,148.992
C03616=1163.331,52.755,-49.663,-179.592,6.172,148.992
C03617=1163.336,52.506,-49.647,-179.594,6.171,148.993
C03618=1163.341,52.256,-49.632,-179.597,6.170,148.993
C03619=1163.345,52.007,-49.616,-179.600,6.169,148.994
C03620=1163.350,51.758,-49.600,-179.602,6.168,148.995
C03621=1163.356,51.508,-49.584,-179.605,6.167,148.995
C03622=1163.361,51.258,-49.568,-179.607,6.166,148.996
C03623=1163.366,51.010,-49.552,-179.610,6.165,148.996
C03624=1163.371,50.760,-49.536,-179.613,6.164,148.997
C03625=1163.376,50.510,-49.521,-179.615,6.163,148.997
C03626=1163.381,50.261,-49.506,-179.618,6.162,148.998
C03627=1163.386,50.012,-49.490,-179.621,6.161,148.999
C03628=1163.390,49.762,-49.473,-179.623,6.160,148.999
C03629=1163.396,49.513,-49.458,-179.626,6.159,149.000
C03630=1163.401,49.263,-49.442,-179.628,6.158,149.000
C03631=1163.405,49.013,-49.427,-179.631,6.157,149.001
C03632=1163.411,48.764,-49.411,-179.633,6.156,149.001
C03633=1163.416,48.515,-49.396,-179.636,6.156,149.002
C03634=1163.420,48.265,-49.379,-179.639,6.154,149.002
C03635=1163.425,48.016,-49.364,-179.641,6.153,149.003
C03636=1163.431,47.767,-49.348,-179.644,6.153,149.003
C03637=1163.435,47.517,-49.332,-179.647,6.151,149.004
C03638=1163.441,47.267,-49.317,-179.649,6.150,149.005
C03639=1163.445,47.018,-49.302,-179.652,6.149,149.005
C03640=1163.451,46.769,-49.286,-179.654,6.148,149.006
C03641=1163.456,46.519,-49.270,-179.657,6.148,149.006
C03642=1163.461,46.269,-49.255,-179.660,6.146,149.007
C03643=1163.466,46.020,-49.240,-179.662,6.146,149.007
C03644=1163.471,45.771,-49.224,-179.665,6.145,149.008
C03645=1163.476,45.521,-49.208,-179.668,6.143,149.009
C03646=1163.480,45.272,-49.192,-179.670,6.143,149.009
C03647=1163.485,45.023,-49.177,-179.673,6.142,149.010
C03648=1163.491,44.773,-49.161,-179.675,6.140,149.010
